LIN {X 0,Y 242.157,Z 688.13,A -85,B 0,C 180,E1 -19275.141,E2 -19275.141} C_VEL
LIN {X 0,Y 242.132,Z 688.251,A -85,B 0,C 180,E1 -19277.962,E2 -19277.962} C_VEL
LIN {X 0,Y 242.388,Z 689.495,A -85,B 0,C 180,E1 -19278.927,E2 -19278.927} C_VEL
LIN {X 0,Y 243.937,Z 692.096,A -85,B 0,C 180,E1 -19280.226,E2 -19280.226} C_VEL
LIN {X 0,Y 247.144,Z 694.46,A -85,B 0,C 180,E1 -19282.354,E2 -19282.354} C_VEL
LIN {X 0,Y 248.695,Z 697.223,A -85,B 0,C 180,E1 -19283.415,E2 -19283.415} C_VEL
LIN {X 0,Y 251.344,Z 699.467,A -85,B 0,C 180,E1 -19284.936,E2 -19284.936} C_VEL
LIN {X 0,Y 251.99,Z 700.132,A -85,B 0,C 180,E1 -19285.297,E2 -19285.297} C_VEL
LIN {X 0,Y 254.265,Z 703.466,A -85,B 0,C 180,E1 -19286.578,E2 -19286.578} C_VEL
LIN {X 0,Y 256.336,Z 705.417,A -85,B 0,C 180,E1 -19287.614,E2 -19287.614} C_VEL
LIN {X 0,Y 258.924,Z 709,A -85,B 0,C 180,E1 -19288.902,E2 -19288.902} C_VEL
LIN {X 0,Y 260.57,Z 710.773,A -85,B 0,C 180,E1 -19289.653,E2 -19289.653} C_VEL
LIN {X 0,Y 263.605,Z 714.655,A -85,B 0,C 180,E1 -19291.005,E2 -19291.005} C_VEL
LIN {X 0,Y 268.675,Z 721.325,A -85,B 0,C 180,E1 -19293.096,E2 -19293.096} C_VEL
LIN {X 0,Y 274.488,Z 729.289,A -85,B 0,C 180,E1 -19295.284,E2 -19295.284} C_VEL
LIN {X 0,Y 282.608,Z 739.443,A -85,B 0,C 180,E1 -19297.978,E2 -19297.978} C_VEL
LIN {X 0,Y 289.117,Z 746.316,A -85,B 0,C 180,E1 -19299.876,E2 -19299.876} C_VEL
LIN {X 0,Y 295.999,Z 752.863,A -85,B 0,C 180,E1 -19301.77,E2 -19301.77} C_VEL
LIN {X 0,Y 303.891,Z 760.01,A -85,B 0,C 180,E1 -19304.075,E2 -19304.075} C_VEL
LIN {X 0,Y 310.616,Z 766.219,A -85,B 0,C 180,E1 -19306.257,E2 -19306.257} C_VEL
LIN {X 0,Y 315.212,Z 770.613,A -85,B 0,C 180,E1 -19307.861,E2 -19307.861} C_VEL
LIN {X 0,Y 320.254,Z 775.282,A -85,B 0,C 180,E1 -19309.758,E2 -19309.758} C_VEL
LIN {X 0,Y 324.928,Z 779.703,A -85,B 0,C 180,E1 -19311.577,E2 -19311.577} C_VEL
LIN {X 0,Y 331.646,Z 785.986,A -85,B 0,C 180,E1 -19314.299,E2 -19314.299} C_VEL
LIN {X 0,Y 335.101,Z 788.959,A -85,B 0,C 180,E1 -19315.743,E2 -19315.743} C_VEL
LIN {X 0,Y 339.882,Z 793.294,A -85,B 0,C 180,E1 -19317.84,E2 -19317.84} C_VEL
LIN {X 0,Y 342.588,Z 795.61,A -85,B 0,C 180,E1 -19319.063,E2 -19319.063} C_VEL
LIN {X 0,Y 346.939,Z 799.679,A -85,B 0,C 180,E1 -19321.138,E2 -19321.138} C_VEL
LIN {X 0,Y 350.25,Z 802.241,A -85,B 0,C 180,E1 -19322.766,E2 -19322.766} C_VEL
LIN {X 0,Y 354.173,Z 806.047,A -85,B 0,C 180,E1 -19324.874,E2 -19324.874} C_VEL
LIN {X 0,Y 358.316,Z 808.916,A -85,B 0,C 180,E1 -19327.197,E2 -19327.197} C_VEL
LIN {X 0,Y 362.043,Z 812.548,A -85,B 0,C 180,E1 -19329.549,E2 -19329.549} C_VEL
LIN {X 0,Y 365.412,Z 815.149,A -85,B 0,C 180,E1 -19331.879,E2 -19331.879} C_VEL
LIN {X 0,Y 368.034,Z 816.748,A -85,B 0,C 180,E1 -19333.849,E2 -19333.849} C_VEL
LIN {X 0,Y 370.527,Z 819.505,A -85,B 0,C 180,E1 -19336.116,E2 -19336.116} C_VEL
LIN {X 0,Y 372.638,Z 821.265,A -85,B 0,C 180,E1 -19338.265,E2 -19338.265} C_VEL
LIN {X 0,Y 374.725,Z 822.511,A -85,B 0,C 180,E1 -19340.809,E2 -19340.809} C_VEL
LIN {X 0,Y 376.488,Z 823.27,A -85,B 0,C 180,E1 -19343.569,E2 -19343.569} C_VEL
LIN {X 0,Y 377.368,Z 823.891,A -85,B 0,C 180,E1 -19345.728,E2 -19345.728} C_VEL
LIN {X 0,Y 377.945,Z 824.103,A -85,B 0,C 180,E1 -19347.869,E2 -19347.869} C_VEL
LIN {X 0,Y 378.148,Z 824.189,A -85,B 0,C 180,E1 -19350,E2 -19350} C_VEL
LIN {X 0,Y 377.944,Z 824.103,A -85,B 0,C 180,E1 -19352.131,E2 -19352.131} C_VEL
LIN {X 0,Y 377.224,Z 823.763,A -85,B 0,C 180,E1 -19354.726,E2 -19354.726} C_VEL
LIN {X 0,Y 376.149,Z 823.23,A -85,B 0,C 180,E1 -19357.007,E2 -19357.007} C_VEL
LIN {X 0,Y 374.33,Z 822.343,A -85,B 0,C 180,E1 -19359.728,E2 -19359.728} C_VEL
LIN {X 0,Y 372.272,Z 820.983,A -85,B 0,C 180,E1 -19362.116,E2 -19362.116} C_VEL
LIN {X 0,Y 369.742,Z 818.743,A -85,B 0,C 180,E1 -19364.631,E2 -19364.631} C_VEL
LIN {X 0,Y 367.379,Z 816.172,A -85,B 0,C 180,E1 -19366.675,E2 -19366.675} C_VEL
LIN {X 0,Y 364.338,Z 814.395,A -85,B 0,C 180,E1 -19368.887,E2 -19368.887} C_VEL
LIN {X 0,Y 360.667,Z 811.337,A -85,B 0,C 180,E1 -19371.326,E2 -19371.326} C_VEL
LIN {X 0,Y 358.319,Z 808.877,A -85,B 0,C 180,E1 -19372.804,E2 -19372.804} C_VEL
LIN {X 0,Y 354.175,Z 806.027,A -85,B 0,C 180,E1 -19375.126,E2 -19375.126} C_VEL
LIN {X 0,Y 350.048,Z 802.014,A -85,B 0,C 180,E1 -19377.342,E2 -19377.342} C_VEL
LIN {X 0,Y 344.973,Z 797.984,A -85,B 0,C 180,E1 -19379.811,E2 -19379.811} C_VEL
LIN {X 0,Y 340.836,Z 794.05,A -85,B 0,C 180,E1 -19381.732,E2 -19381.732} C_VEL
LIN {X 0,Y 335.827,Z 789.683,A -85,B 0,C 180,E1 -19383.943,E2 -19383.943} C_VEL
LIN {X 0,Y 332.449,Z 786.584,A -85,B 0,C 180,E1 -19385.377,E2 -19385.377} C_VEL
LIN {X 0,Y 327.426,Z 782.051,A -85,B 0,C 180,E1 -19387.423,E2 -19387.423} C_VEL
LIN {X 0,Y 324.201,Z 779.091,A -85,B 0,C 180,E1 -19388.703,E2 -19388.703} C_VEL
LIN {X 0,Y 319.113,Z 774.042,A -85,B 0,C 180,E1 -19390.689,E2 -19390.689} C_VEL
LIN {X 0,Y 314.019,Z 769.41,A -85,B 0,C 180,E1 -19392.567,E2 -19392.567} C_VEL
LIN {X 0,Y 309.624,Z 765.385,A -85,B 0,C 180,E1 -19394.072,E2 -19394.072} C_VEL
LIN {X 0,Y 303.772,Z 759.909,A -85,B 0,C 180,E1 -19395.962,E2 -19395.962} C_VEL
LIN {X 0,Y 298.163,Z 754.652,A -85,B 0,C 180,E1 -19397.626,E2 -19397.626} C_VEL
LIN {X 0,Y 291.81,Z 748.998,A -85,B 0,C 180,E1 -19399.386,E2 -19399.386} C_VEL
LIN {X 0,Y 283.81,Z 740.718,A -85,B 0,C 180,E1 -19401.658,E2 -19401.658} C_VEL
LIN {X 0,Y 278.243,Z 734.184,A -85,B 0,C 180,E1 -19403.421,E2 -19403.421} C_VEL
LIN {X 0,Y 269.096,Z 721.878,A -85,B 0,C 180,E1 -19406.739,E2 -19406.739} C_VEL
LIN {X 0,Y 266.598,Z 718.603,A -85,B 0,C 180,E1 -19407.736,E2 -19407.736} C_VEL
LIN {X 0,Y 263.457,Z 714.51,A -85,B 0,C 180,E1 -19409.057,E2 -19409.057} C_VEL
LIN {X 0,Y 260.385,Z 710.48,A -85,B 0,C 180,E1 -19410.435,E2 -19410.435} C_VEL
LIN {X 0,Y 256.965,Z 706.492,A -85,B 0,C 180,E1 -19412.054,E2 -19412.054} C_VEL
LIN {X 0,Y 255.896,Z 704.836,A -85,B 0,C 180,E1 -19412.612,E2 -19412.612} C_VEL
LIN {X 0,Y 253.226,Z 702.224,A -85,B 0,C 180,E1 -19413.979,E2 -19413.979} C_VEL
LIN {X 0,Y 251.561,Z 699.597,A -85,B 0,C 180,E1 -19414.948,E2 -19414.948} C_VEL
LIN {X 0,Y 248.847,Z 697.414,A -85,B 0,C 180,E1 -19416.49,E2 -19416.49} C_VEL
LIN {X 0,Y 246.704,Z 693.991,A -85,B 0,C 180,E1 -19417.934,E2 -19417.934} C_VEL
LIN {X 0,Y 243.937,Z 692.096,A -85,B 0,C 180,E1 -19419.774,E2 -19419.774} C_VEL
LIN {X 0,Y 242.353,Z 689.417,A -85,B 0,C 180,E1 -19421.125,E2 -19421.125} C_VEL
LIN {X 0,Y 242.133,Z 688.246,A -85,B 0,C 180,E1 -19422.093,E2 -19422.093} C_VEL
LIN {X 0,Y 242.156,Z 688.106,A -85,B 0,C 180,E1 -19426.575,E2 -19426.575} C_VEL
LIN {X 0,Y 242.419,Z 688.073,A -85,B 0,C 180,E1 -19431.666,E2 -19431.666} C_VEL
LIN {X 0,Y 242.256,Z 688.12,A -85,B 0,C 180,E1 -19435.008,E2 -19435.008} C_VEL
LIN {X 0,Y 242.631,Z 688.05,A -85,B 0,C 180,E1 -19438.341,E2 -19438.341} C_VEL
LIN {X 0,Y 242.631,Z 688.052,A -85,B 0,C 180,E1 -19441.66,E2 -19441.66} C_VEL
LIN {X 0,Y 242.427,Z 688.078,A -85,B 0,C 180,E1 -19446.659,E2 -19446.659} C_VEL
LIN {X 0,Y 242.309,Z 688.104,A -85,B 0,C 180,E1 -19450.022,E2 -19450.022} C_VEL
LIN {X 0,Y 242.151,Z 688.127,A -85,B 0,C 180,E1 -19455.142,E2 -19455.142} C_VEL
LIN {X 0,Y 242.154,Z 688.429,A -85,B 0,C 180,E1 -19457.743,E2 -19457.743} C_VEL
LIN {X 0,Y 242.453,Z 689.706,A -85,B 0,C 180,E1 -19458.594,E2 -19458.594} C_VEL
LIN {X 0,Y 243.896,Z 692.084,A -85,B 0,C 180,E1 -19459.791,E2 -19459.791} C_VEL
LIN {X 0,Y 246.644,Z 693.971,A -85,B 0,C 180,E1 -19461.623,E2 -19461.623} C_VEL
LIN {X 0,Y 247.502,Z 695.283,A -85,B 0,C 180,E1 -19462.211,E2 -19462.211} C_VEL
LIN {X 0,Y 249.266,Z 697.887,A -85,B 0,C 180,E1 -19463.359,E2 -19463.359} C_VEL
LIN {X 0,Y 251.914,Z 700.026,A -85,B 0,C 180,E1 -19464.846,E2 -19464.846} C_VEL
LIN {X 0,Y 254.117,Z 703.305,A -85,B 0,C 180,E1 -19466.094,E2 -19466.094} C_VEL
LIN {X 0,Y 256.371,Z 705.449,A -85,B 0,C 180,E1 -19467.224,E2 -19467.224} C_VEL
LIN {X 0,Y 259.014,Z 709.076,A -85,B 0,C 180,E1 -19468.535,E2 -19468.535} C_VEL
LIN {X 0,Y 260.601,Z 710.841,A -85,B 0,C 180,E1 -19469.262,E2 -19469.262} C_VEL
LIN {X 0,Y 263.715,Z 714.755,A -85,B 0,C 180,E1 -19470.643,E2 -19470.643} C_VEL
LIN {X 0,Y 268.241,Z 721.279,A -85,B 0,C 180,E1 -19472.543,E2 -19472.543} C_VEL
LIN {X 0,Y 272.38,Z 727.881,A -85,B 0,C 180,E1 -19474.176,E2 -19474.176} C_VEL
LIN {X 0,Y 279.24,Z 739.541,A -85,B 0,C 180,E1 -19476.675,E2 -19476.675} C_VEL
LIN {X 0,Y 286.08,Z 752.594,A -85,B 0,C 180,E1 -19478.974,E2 -19478.974} C_VEL
LIN {X 0,Y 292.085,Z 765.049,A -85,B 0,C 180,E1 -19480.857,E2 -19480.857} C_VEL
LIN {X 0,Y 296.083,Z 774.289,A -85,B 0,C 180,E1 -19482.065,E2 -19482.065} C_VEL
LIN {X 0,Y 295.264,Z 789.935,A -85,B 0,C 180,E1 -19482.443,E2 -19482.443} C_VEL
LIN {X 0,Y 294.474,Z 795.788,A -85,B 0,C 180,E1 -19482.482,E2 -19482.482} C_VEL
LIN {X 0,Y 289.416,Z 814.875,A -85,B 0,C 180,E1 -19482.08,E2 -19482.08} C_VEL
LIN {X 0,Y 288.604,Z 820.73,A -85,B 0,C 180,E1 -19482.114,E2 -19482.114} C_VEL
LIN {X 0,Y 284.395,Z 890.144,A -85,B 0,C 180,E1 -19483.772,E2 -19483.772} C_VEL
LIN {X 0,Y 283.091,Z 902.745,A -85,B 0,C 180,E1 -19484.196,E2 -19484.196} C_VEL
LIN {X 0,Y 281.233,Z 915.218,A -85,B 0,C 180,E1 -19484.73,E2 -19484.73} C_VEL
LIN {X 0,Y 278.913,Z 927.393,A -85,B 0,C 180,E1 -19485.382,E2 -19485.382} C_VEL
LIN {X 0,Y 276.549,Z 938.778,A -85,B 0,C 180,E1 -19486.172,E2 -19486.172} C_VEL
LIN {X 0,Y 273.265,Z 952.009,A -85,B 0,C 180,E1 -19487.288,E2 -19487.288} C_VEL
LIN {X 0,Y 270.044,Z 963.302,A -85,B 0,C 180,E1 -19488.423,E2 -19488.423} C_VEL
LIN {X 0,Y 266.166,Z 975.709,A -85,B 0,C 180,E1 -19489.935,E2 -19489.935} C_VEL
LIN {X 0,Y 262.462,Z 986.529,A -85,B 0,C 180,E1 -19491.497,E2 -19491.497} C_VEL
LIN {X 0,Y 258.484,Z 997.021,A -85,B 0,C 180,E1 -19493.263,E2 -19493.263} C_VEL
LIN {X 0,Y 254.908,Z 1006.289,A -85,B 0,C 180,E1 -19495.105,E2 -19495.105} C_VEL
LIN {X 0,Y 250.75,Z 1016.429,A -85,B 0,C 180,E1 -19497.482,E2 -19497.482} C_VEL
LIN {X 0,Y 247.32,Z 1024.542,A -85,B 0,C 180,E1 -19499.71,E2 -19499.71} C_VEL
LIN {X 0,Y 243.66,Z 1033.143,A -85,B 0,C 180,E1 -19502.517,E2 -19502.517} C_VEL
LIN {X 0,Y 240.85,Z 1039.875,A -85,B 0,C 180,E1 -19505.114,E2 -19505.114} C_VEL
LIN {X 0,Y 238.008,Z 1046.841,A -85,B 0,C 180,E1 -19508.34,E2 -19508.34} C_VEL
LIN {X 0,Y 236.243,Z 1051.496,A -85,B 0,C 180,E1 -19510.899,E2 -19510.899} C_VEL
LIN {X 0,Y 234.564,Z 1056.604,A -85,B 0,C 180,E1 -19514.357,E2 -19514.357} C_VEL
LIN {X 0,Y 233.371,Z 1060.609,A -85,B 0,C 180,E1 -19517.831,E2 -19517.831} C_VEL
LIN {X 0,Y 232.842,Z 1063.577,A -85,B 0,C 180,E1 -19521.32,E2 -19521.32} C_VEL
LIN {X 0,Y 232.7,Z 1064.768,A -85,B 0,C 180,E1 -19523.061,E2 -19523.061} C_VEL
LIN {X 0,Y 232.651,Z 1066.246,A -85,B 0,C 180,E1 -19526.536,E2 -19526.536} C_VEL
LIN {X 0,Y 232.801,Z 1066.741,A -85,B 0,C 180,E1 -19530,E2 -19530} C_VEL
LIN {X 0,Y 232.651,Z 1066.246,A -85,B 0,C 180,E1 -19533.464,E2 -19533.464} C_VEL
LIN {X 0,Y 232.7,Z 1064.768,A -85,B 0,C 180,E1 -19536.939,E2 -19536.939} C_VEL
LIN {X 0,Y 233.04,Z 1062.289,A -85,B 0,C 180,E1 -19540.425,E2 -19540.425} C_VEL
LIN {X 0,Y 234.206,Z 1057.693,A -85,B 0,C 180,E1 -19544.777,E2 -19544.777} C_VEL
LIN {X 0,Y 235.787,Z 1052.848,A -85,B 0,C 180,E1 -19548.238,E2 -19548.238} C_VEL
LIN {X 0,Y 237.391,Z 1048.465,A -85,B 0,C 180,E1 -19550.809,E2 -19550.809} C_VEL
LIN {X 0,Y 239.44,Z 1043.402,A -85,B 0,C 180,E1 -19553.343,E2 -19553.343} C_VEL
LIN {X 0,Y 242.248,Z 1036.477,A -85,B 0,C 180,E1 -19556.258,E2 -19556.258} C_VEL
LIN {X 0,Y 245.703,Z 1028.382,A -85,B 0,C 180,E1 -19559.094,E2 -19559.094} C_VEL
LIN {X 0,Y 249.164,Z 1020.417,A -85,B 0,C 180,E1 -19561.453,E2 -19561.453} C_VEL
LIN {X 0,Y 252.896,Z 1011.305,A -85,B 0,C 180,E1 -19563.765,E2 -19563.765} C_VEL
LIN {X 0,Y 256.333,Z 1002.739,A -85,B 0,C 180,E1 -19565.634,E2 -19565.634} C_VEL
LIN {X 0,Y 260.727,Z 990.874,A -85,B 0,C 180,E1 -19567.823,E2 -19567.823} C_VEL
LIN {X 0,Y 264.497,Z 980.719,A -85,B 0,C 180,E1 -19569.373,E2 -19569.373} C_VEL
LIN {X 0,Y 268.315,Z 969.054,A -85,B 0,C 180,E1 -19570.905,E2 -19570.905} C_VEL
LIN {X 0,Y 271.869,Z 957.033,A -85,B 0,C 180,E1 -19572.229,E2 -19572.229} C_VEL
LIN {X 0,Y 275.13,Z 944.719,A -85,B 0,C 180,E1 -19573.352,E2 -19573.352} C_VEL
LIN {X 0,Y 277.951,Z 932.178,A -85,B 0,C 180,E1 -19574.305,E2 -19574.305} C_VEL
LIN {X 0,Y 280.57,Z 918.763,A -85,B 0,C 180,E1 -19575.104,E2 -19575.104} C_VEL
LIN {X 0,Y 282.658,Z 905.869,A -85,B 0,C 180,E1 -19575.691,E2 -19575.691} C_VEL
LIN {X 0,Y 284.256,Z 892.458,A -85,B 0,C 180,E1 -19576.149,E2 -19576.149} C_VEL
LIN {X 0,Y 285.97,Z 865.198,A -85,B 0,C 180,E1 -19576.851,E2 -19576.851} C_VEL
LIN {X 0,Y 291.182,Z 777.985,A -85,B 0,C 180,E1 -19578.872,E2 -19578.872} C_VEL
LIN {X 0,Y 291.068,Z 776.493,A -85,B 0,C 180,E1 -19578.952,E2 -19578.952} C_VEL
LIN {X 0,Y 285.259,Z 763.336,A -85,B 0,C 180,E1 -19580.809,E2 -19580.809} C_VEL
LIN {X 0,Y 278.575,Z 749.866,A -85,B 0,C 180,E1 -19583.074,E2 -19583.074} C_VEL
LIN {X 0,Y 273.098,Z 739.77,A -85,B 0,C 180,E1 -19585.069,E2 -19585.069} C_VEL
LIN {X 0,Y 266.936,Z 729.437,A -85,B 0,C 180,E1 -19587.495,E2 -19587.495} C_VEL
LIN {X 0,Y 263.033,Z 723.353,A -85,B 0,C 180,E1 -19589.158,E2 -19589.158} C_VEL
LIN {X 0,Y 260.683,Z 720.268,A -85,B 0,C 180,E1 -19590.193,E2 -19590.193} C_VEL
LIN {X 0,Y 257.341,Z 715.903,A -85,B 0,C 180,E1 -19591.757,E2 -19591.757} C_VEL
LIN {X 0,Y 254.259,Z 711.919,A -85,B 0,C 180,E1 -19593.309,E2 -19593.309} C_VEL
LIN {X 0,Y 250.599,Z 707.706,A -85,B 0,C 180,E1 -19595.289,E2 -19595.289} C_VEL
LIN {X 0,Y 249.582,Z 706.174,A -85,B 0,C 180,E1 -19595.901,E2 -19595.901} C_VEL
LIN {X 0,Y 246.769,Z 703.584,A -85,B 0,C 180,E1 -19597.581,E2 -19597.581} C_VEL
LIN {X 0,Y 245.071,Z 700.739,A -85,B 0,C 180,E1 -19598.777,E2 -19598.777} C_VEL
LIN {X 0,Y 242.377,Z 698.784,A -85,B 0,C 180,E1 -19600.631,E2 -19600.631} C_VEL
LIN {X 0,Y 240.648,Z 695.967,A -85,B 0,C 180,E1 -19602.087,E2 -19602.087} C_VEL
LIN {X 0,Y 239.897,Z 694.934,A -85,B 0,C 180,E1 -19602.745,E2 -19602.745} C_VEL
LIN {X 0,Y 236.953,Z 692.981,A -85,B 0,C 180,E1 -19605.397,E2 -19605.397} C_VEL
LIN {X 0,Y 235.329,Z 690.078,A -85,B 0,C 180,E1 -19607.495,E2 -19607.495} C_VEL
LIN {X 0,Y 235.168,Z 689.024,A -85,B 0,C 180,E1 -19608.962,E2 -19608.962} C_VEL
LIN {X 0,Y 235.371,Z 688.951,A -85,B 0,C 180,E1 -19611.413,E2 -19611.413} C_VEL
LIN {X 0,Y 235.398,Z 688.95,A -85,B 0,C 180,E1 -19613.141,E2 -19613.141} C_VEL
LIN {X 0,Y 235.59,Z 688.926,A -85,B 0,C 180,E1 -19618.29,E2 -19618.29} C_VEL
LIN {X 0,Y 235.59,Z 688.925,A -85,B 0,C 180,E1 -19621.709,E2 -19621.709} C_VEL
LIN {X 0,Y 235.397,Z 688.951,A -85,B 0,C 180,E1 -19626.858,E2 -19626.858} C_VEL
LIN {X 0,Y 235.232,Z 689.005,A -85,B 0,C 180,E1 -19630.326,E2 -19630.326} C_VEL
LIN {X 0,Y 235.194,Z 689.499,A -85,B 0,C 180,E1 -19632.292,E2 -19632.292} C_VEL
LIN {X 0,Y 235.642,Z 690.924,A -85,B 0,C 180,E1 -19633.474,E2 -19633.474} C_VEL
LIN {X 0,Y 237.185,Z 693.203,A -85,B 0,C 180,E1 -19635.246,E2 -19635.246} C_VEL
LIN {X 0,Y 240.413,Z 695.413,A -85,B 0,C 180,E1 -19638.095,E2 -19638.095} C_VEL
LIN {X 0,Y 242.289,Z 698.654,A -85,B 0,C 180,E1 -19639.706,E2 -19639.706} C_VEL
LIN {X 0,Y 244.989,Z 700.698,A -85,B 0,C 180,E1 -19641.578,E2 -19641.578} C_VEL
LIN {X 0,Y 247.688,Z 704.621,A -85,B 0,C 180,E1 -19643.405,E2 -19643.405} C_VEL
LIN {X 0,Y 250.035,Z 706.686,A -85,B 0,C 180,E1 -19644.77,E2 -19644.77} C_VEL
LIN {X 0,Y 252.548,Z 710.161,A -85,B 0,C 180,E1 -19646.21,E2 -19646.21} C_VEL
LIN {X 0,Y 254.313,Z 712.015,A -85,B 0,C 180,E1 -19647.127,E2 -19647.127} C_VEL
LIN {X 0,Y 257.121,Z 715.679,A -85,B 0,C 180,E1 -19648.546,E2 -19648.546} C_VEL
LIN {X 0,Y 258.462,Z 717.383,A -85,B 0,C 180,E1 -19649.188,E2 -19649.188} C_VEL
LIN {X 0,Y 262.751,Z 722.957,A -85,B 0,C 180,E1 -19651.126,E2 -19651.126} C_VEL
LIN {X 0,Y 266.457,Z 727.884,A -85,B 0,C 180,E1 -19652.675,E2 -19652.675} C_VEL
LIN {X 0,Y 279.488,Z 745.151,A -85,B 0,C 180,E1 -19657.384,E2 -19657.384} C_VEL
LIN {X 0,Y 286.696,Z 752.785,A -85,B 0,C 180,E1 -19659.54,E2 -19659.54} C_VEL
LIN {X 0,Y 293.599,Z 759.313,A -85,B 0,C 180,E1 -19661.43,E2 -19661.43} C_VEL
LIN {X 0,Y 300.628,Z 765.685,A -85,B 0,C 180,E1 -19663.455,E2 -19663.455} C_VEL
LIN {X 0,Y 304.805,Z 769.406,A -85,B 0,C 180,E1 -19664.728,E2 -19664.728} C_VEL
LIN {X 0,Y 309.685,Z 773.681,A -85,B 0,C 180,E1 -19666.306,E2 -19666.306} C_VEL
LIN {X 0,Y 315.306,Z 779.062,A -85,B 0,C 180,E1 -19668.282,E2 -19668.282} C_VEL
LIN {X 0,Y 319.999,Z 783.569,A -85,B 0,C 180,E1 -19670.062,E2 -19670.062} C_VEL
LIN {X 0,Y 325.699,Z 788.7,A -85,B 0,C 180,E1 -19672.28,E2 -19672.28} C_VEL
LIN {X 0,Y 330.659,Z 793.216,A -85,B 0,C 180,E1 -19674.297,E2 -19674.297} C_VEL
LIN {X 0,Y 333.474,Z 795.703,A -85,B 0,C 180,E1 -19675.473,E2 -19675.473} C_VEL
LIN {X 0,Y 338.278,Z 800.003,A -85,B 0,C 180,E1 -19677.547,E2 -19677.547} C_VEL
LIN {X 0,Y 340.875,Z 802.2,A -85,B 0,C 180,E1 -19678.714,E2 -19678.714} C_VEL
LIN {X 0,Y 345.38,Z 806.398,A -85,B 0,C 180,E1 -19680.847,E2 -19680.847} C_VEL
LIN {X 0,Y 348.716,Z 808.932,A -85,B 0,C 180,E1 -19682.469,E2 -19682.469} C_VEL
LIN {X 0,Y 352.697,Z 812.745,A -85,B 0,C 180,E1 -19684.577,E2 -19684.577} C_VEL
LIN {X 0,Y 356.872,Z 815.691,A -85,B 0,C 180,E1 -19686.88,E2 -19686.88} C_VEL
LIN {X 0,Y 360.806,Z 819.411,A -85,B 0,C 180,E1 -19689.334,E2 -19689.334} C_VEL
LIN {X 0,Y 364.226,Z 822.049,A -85,B 0,C 180,E1 -19691.676,E2 -19691.676} C_VEL
LIN {X 0,Y 366.994,Z 823.751,A -85,B 0,C 180,E1 -19693.725,E2 -19693.725} C_VEL
LIN {X 0,Y 369.473,Z 826.446,A -85,B 0,C 180,E1 -19695.952,E2 -19695.952} C_VEL
LIN {X 0,Y 371.492,Z 828.14,A -85,B 0,C 180,E1 -19697.989,E2 -19697.989} C_VEL
LIN {X 0,Y 373.441,Z 829.38,A -85,B 0,C 180,E1 -19700.249,E2 -19700.249} C_VEL
LIN {X 0,Y 375.282,Z 830.27,A -85,B 0,C 180,E1 -19702.993,E2 -19702.993} C_VEL
LIN {X 0,Y 376.498,Z 830.932,A -85,B 0,C 180,E1 -19705.718,E2 -19705.718} C_VEL
LIN {X 0,Y 377.076,Z 831.149,A -85,B 0,C 180,E1 -19707.864,E2 -19707.864} C_VEL
LIN {X 0,Y 377.283,Z 831.235,A -85,B 0,C 180,E1 -19710,E2 -19710} C_VEL
LIN {X 0,Y 377.076,Z 831.148,A -85,B 0,C 180,E1 -19712.136,E2 -19712.136} C_VEL
LIN {X 0,Y 376.354,Z 830.811,A -85,B 0,C 180,E1 -19714.737,E2 -19714.737} C_VEL
LIN {X 0,Y 375.104,Z 830.173,A -85,B 0,C 180,E1 -19717.299,E2 -19717.299} C_VEL
LIN {X 0,Y 373.441,Z 829.385,A -85,B 0,C 180,E1 -19719.751,E2 -19719.751} C_VEL
LIN {X 0,Y 371.365,Z 828.015,A -85,B 0,C 180,E1 -19722.146,E2 -19722.146} C_VEL
LIN {X 0,Y 368.91,Z 825.922,A -85,B 0,C 180,E1 -19724.58,E2 -19724.58} C_VEL
LIN {X 0,Y 366.201,Z 823.109,A -85,B 0,C 180,E1 -19726.89,E2 -19726.89} C_VEL
LIN {X 0,Y 362.98,Z 821.155,A -85,B 0,C 180,E1 -19729.217,E2 -19729.217} C_VEL
LIN {X 0,Y 359.096,Z 817.848,A -85,B 0,C 180,E1 -19731.759,E2 -19731.759} C_VEL
LIN {X 0,Y 356.973,Z 815.726,A -85,B 0,C 180,E1 -19733.061,E2 -19733.061} C_VEL
LIN {X 0,Y 352.563,Z 812.65,A -85,B 0,C 180,E1 -19735.495,E2 -19735.495} C_VEL
LIN {X 0,Y 347.543,Z 807.97,A -85,B 0,C 180,E1 -19738.112,E2 -19738.112} C_VEL
LIN {X 0,Y 343.037,Z 804.349,A -85,B 0,C 180,E1 -19740.266,E2 -19740.266} C_VEL
LIN {X 0,Y 339.196,Z 800.725,A -85,B 0,C 180,E1 -19742.037,E2 -19742.037} C_VEL
LIN {X 0,Y 334.098,Z 796.312,A -85,B 0,C 180,E1 -19744.261,E2 -19744.261} C_VEL
LIN {X 0,Y 330.812,Z 793.323,A -85,B 0,C 180,E1 -19745.642,E2 -19745.642} C_VEL
LIN {X 0,Y 325.496,Z 788.535,A -85,B 0,C 180,E1 -19747.801,E2 -19747.801} C_VEL
LIN {X 0,Y 318.755,Z 782.313,A -85,B 0,C 180,E1 -19750.423,E2 -19750.423} C_VEL
LIN {X 0,Y 315.079,Z 778.87,A -85,B 0,C 180,E1 -19751.799,E2 -19751.799} C_VEL
LIN {X 0,Y 308.446,Z 772.688,A -85,B 0,C 180,E1 -19754.104,E2 -19754.104} C_VEL
LIN {X 0,Y 301.432,Z 766.329,A -85,B 0,C 180,E1 -19756.309,E2 -19756.309} C_VEL
LIN {X 0,Y 296.413,Z 761.822,A -85,B 0,C 180,E1 -19757.777,E2 -19757.777} C_VEL
LIN {X 0,Y 288.735,Z 754.866,A -85,B 0,C 180,E1 -19759.89,E2 -19759.89} C_VEL
LIN {X 0,Y 281.034,Z 746.827,A -85,B 0,C 180,E1 -19762.134,E2 -19762.134} C_VEL
LIN {X 0,Y 275.221,Z 739.886,A -85,B 0,C 180,E1 -19764.033,E2 -19764.033} C_VEL
LIN {X 0,Y 264.577,Z 725.223,A -85,B 0,C 180,E1 -19768.105,E2 -19768.105} C_VEL
LIN {X 0,Y 260.8,Z 720.394,A -85,B 0,C 180,E1 -19769.735,E2 -19769.735} C_VEL
LIN {X 0,Y 257.235,Z 715.776,A -85,B 0,C 180,E1 -19771.401,E2 -19771.401} C_VEL
LIN {X 0,Y 254.398,Z 712.153,A -85,B 0,C 180,E1 -19772.827,E2 -19772.827} C_VEL
LIN {X 0,Y 253.263,Z 710.813,A -85,B 0,C 180,E1 -19773.419,E2 -19773.419} C_VEL
LIN {X 0,Y 250.554,Z 707.612,A -85,B 0,C 180,E1 -19774.91,E2 -19774.91} C_VEL
LIN {X 0,Y 249.639,Z 706.166,A -85,B 0,C 180,E1 -19775.465,E2 -19775.465} C_VEL
LIN {X 0,Y 246.853,Z 703.681,A -85,B 0,C 180,E1 -19777.121,E2 -19777.121} C_VEL
LIN {X 0,Y 244.989,Z 700.698,A -85,B 0,C 180,E1 -19778.422,E2 -19778.422} C_VEL
LIN {X 0,Y 242.291,Z 698.641,A -85,B 0,C 180,E1 -19780.294,E2 -19780.294} C_VEL
LIN {X 0,Y 240.575,Z 695.76,A -85,B 0,C 180,E1 -19781.753,E2 -19781.753} C_VEL
LIN {X 0,Y 239.683,Z 694.844,A -85,B 0,C 180,E1 -19782.51,E2 -19782.51} C_VEL
LIN {X 0,Y 236.785,Z 692.785,A -85,B 0,C 180,E1 -19785.168,E2 -19785.168} C_VEL
LIN {X 0,Y 235.347,Z 690.143,A -85,B 0,C 180,E1 -19787.058,E2 -19787.058} C_VEL
LIN {X 0,Y 235.176,Z 689.072,A -85,B 0,C 180,E1 -19788.582,E2 -19788.582} C_VEL
LIN {X 0,Y 235.369,Z 688.952,A -85,B 0,C 180,E1 -19791.414,E2 -19791.414} C_VEL
LIN {X 0,Y 235.396,Z 688.949,A -85,B 0,C 180,E1 -19793.142,E2 -19793.142} C_VEL
LIN {X 0,Y 235.59,Z 688.926,A -85,B 0,C 180,E1 -19798.291,E2 -19798.291} C_VEL
LIN {X 0,Y 235.59,Z 688.928,A -85,B 0,C 180,E1 -19801.71,E2 -19801.71} C_VEL
LIN {X 0,Y 235.398,Z 688.951,A -85,B 0,C 180,E1 -19806.859,E2 -19806.859} C_VEL
LIN {X 0,Y 235.2,Z 689.043,A -85,B 0,C 180,E1 -19810.764,E2 -19810.764} C_VEL
LIN {X 0,Y 235.238,Z 689.626,A -85,B 0,C 180,E1 -19812.072,E2 -19812.072} C_VEL
LIN {X 0,Y 235.938,Z 691.525,A -85,B 0,C 180,E1 -19813.457,E2 -19813.457} C_VEL
LIN {X 0,Y 237.788,Z 693.718,A -85,B 0,C 180,E1 -19815.427,E2 -19815.427} C_VEL
LIN {X 0,Y 240.378,Z 695.377,A -85,B 0,C 180,E1 -19817.658,E2 -19817.658} C_VEL
LIN {X 0,Y 242.119,Z 698.486,A -85,B 0,C 180,E1 -19819.17,E2 -19819.17} C_VEL
LIN {X 0,Y 244.692,Z 700.576,A -85,B 0,C 180,E1 -19820.983,E2 -19820.983} C_VEL
LIN {X 0,Y 245.385,Z 701.183,A -85,B 0,C 180,E1 -19821.444,E2 -19821.444} C_VEL
LIN {X 0,Y 247.178,Z 704.096,A -85,B 0,C 180,E1 -19822.683,E2 -19822.683} C_VEL
LIN {X 0,Y 250.063,Z 706.745,A -85,B 0,C 180,E1 -19824.381,E2 -19824.381} C_VEL
LIN {X 0,Y 252.489,Z 710.106,A -85,B 0,C 180,E1 -19825.772,E2 -19825.772} C_VEL
LIN {X 0,Y 254.343,Z 712.062,A -85,B 0,C 180,E1 -19826.736,E2 -19826.736} C_VEL
LIN {X 0,Y 257.459,Z 716.038,A -85,B 0,C 180,E1 -19828.299,E2 -19828.299} C_VEL
LIN {X 0,Y 262.541,Z 722.671,A -85,B 0,C 180,E1 -19830.627,E2 -19830.627} C_VEL
LIN {X 0,Y 265.549,Z 727.214,A -85,B 0,C 180,E1 -19831.925,E2 -19831.925} C_VEL
LIN {X 0,Y 270.85,Z 735.879,A -85,B 0,C 180,E1 -19834.071,E2 -19834.071} C_VEL
LIN {X 0,Y 277.073,Z 747.03,A -85,B 0,C 180,E1 -19836.393,E2 -19836.393} C_VEL
LIN {X 0,Y 283.438,Z 759.57,A -85,B 0,C 180,E1 -19838.592,E2 -19838.592} C_VEL
LIN {X 0,Y 289.231,Z 772.137,A -85,B 0,C 180,E1 -19840.469,E2 -19840.469} C_VEL
LIN {X 0,Y 291.187,Z 776.785,A -85,B 0,C 180,E1 -19841.085,E2 -19841.085} C_VEL
LIN {X 0,Y 288.604,Z 820.73,A -85,B 0,C 180,E1 -19842.114,E2 -19842.114} C_VEL
LIN {X 0,Y 287.794,Z 826.586,A -85,B 0,C 180,E1 -19842.15,E2 -19842.15} C_VEL
LIN {X 0,Y 282.774,Z 845.685,A -85,B 0,C 180,E1 -19841.738,E2 -19841.738} C_VEL
LIN {X 0,Y 281.985,Z 851.539,A -85,B 0,C 180,E1 -19841.778,E2 -19841.778} C_VEL
LIN {X 0,Y 279.451,Z 890.753,A -85,B 0,C 180,E1 -19842.743,E2 -19842.743} C_VEL
LIN {X 0,Y 278.04,Z 903.623,A -85,B 0,C 180,E1 -19843.188,E2 -19843.188} C_VEL
LIN {X 0,Y 276.08,Z 916.12,A -85,B 0,C 180,E1 -19843.738,E2 -19843.738} C_VEL
LIN {X 0,Y 273.637,Z 928.383,A -85,B 0,C 180,E1 -19844.414,E2 -19844.414} C_VEL
LIN {X 0,Y 270.963,Z 940.552,A -85,B 0,C 180,E1 -19845.29,E2 -19845.29} C_VEL
LIN {X 0,Y 268.073,Z 951.803,A -85,B 0,C 180,E1 -19846.255,E2 -19846.255} C_VEL
LIN {X 0,Y 264.273,Z 964.533,A -85,B 0,C 180,E1 -19847.562,E2 -19847.562} C_VEL
LIN {X 0,Y 260.621,Z 975.811,A -85,B 0,C 180,E1 -19848.965,E2 -19848.965} C_VEL
LIN {X 0,Y 256.922,Z 986.323,A -85,B 0,C 180,E1 -19850.507,E2 -19850.507} C_VEL
LIN {X 0,Y 252.775,Z 996.813,A -85,B 0,C 180,E1 -19852.291,E2 -19852.291} C_VEL
LIN {X 0,Y 249.057,Z 1006.082,A -85,B 0,C 180,E1 -19854.16,E2 -19854.16} C_VEL
LIN {X 0,Y 244.839,Z 1015.845,A -85,B 0,C 180,E1 -19856.47,E2 -19856.47} C_VEL
LIN {X 0,Y 241.125,Z 1024.333,A -85,B 0,C 180,E1 -19858.846,E2 -19858.846} C_VEL
LIN {X 0,Y 237.284,Z 1032.934,A -85,B 0,C 180,E1 -19861.713,E2 -19861.713} C_VEL
LIN {X 0,Y 234.061,Z 1040.26,A -85,B 0,C 180,E1 -19864.636,E2 -19864.636} C_VEL
LIN {X 0,Y 231.333,Z 1046.633,A -85,B 0,C 180,E1 -19867.682,E2 -19867.682} C_VEL
LIN {X 0,Y 229.454,Z 1051.288,A -85,B 0,C 180,E1 -19870.311,E2 -19870.311} C_VEL
LIN {X 0,Y 227.632,Z 1056.395,A -85,B 0,C 180,E1 -19873.867,E2 -19873.867} C_VEL
LIN {X 0,Y 226.366,Z 1060.402,A -85,B 0,C 180,E1 -19877.448,E2 -19877.448} C_VEL
LIN {X 0,Y 225.761,Z 1063.37,A -85,B 0,C 180,E1 -19881.046,E2 -19881.046} C_VEL
LIN {X 0,Y 225.61,Z 1064.562,A -85,B 0,C 180,E1 -19882.842,E2 -19882.842} C_VEL
LIN {X 0,Y 225.549,Z 1066.04,A -85,B 0,C 180,E1 -19886.427,E2 -19886.427} C_VEL
LIN {X 0,Y 225.714,Z 1066.536,A -85,B 0,C 180,E1 -19890,E2 -19890} C_VEL
LIN {X 0,Y 225.554,Z 1065.725,A -85,B 0,C 180,E1 -19894.378,E2 -19894.378} C_VEL
LIN {X 0,Y 225.61,Z 1064.562,A -85,B 0,C 180,E1 -19897.158,E2 -19897.158} C_VEL
LIN {X 0,Y 226.005,Z 1062.082,A -85,B 0,C 180,E1 -19900.753,E2 -19900.753} C_VEL
LIN {X 0,Y 227.264,Z 1057.485,A -85,B 0,C 180,E1 -19905.239,E2 -19905.239} C_VEL
LIN {X 0,Y 228.444,Z 1053.989,A -85,B 0,C 180,E1 -19907.917,E2 -19907.917} C_VEL
LIN {X 0,Y 230.665,Z 1048.256,A -85,B 0,C 180,E1 -19911.445,E2 -19911.445} C_VEL
LIN {X 0,Y 232.826,Z 1043.193,A -85,B 0,C 180,E1 -19914.048,E2 -19914.048} C_VEL
LIN {X 0,Y 235.796,Z 1036.268,A -85,B 0,C 180,E1 -19917.034,E2 -19917.034} C_VEL
LIN {X 0,Y 239.444,Z 1028.174,A -85,B 0,C 180,E1 -19919.931,E2 -19919.931} C_VEL
LIN {X 0,Y 243.025,Z 1020.208,A -85,B 0,C 180,E1 -19922.343,E2 -19922.343} C_VEL
LIN {X 0,Y 246.926,Z 1011.096,A -85,B 0,C 180,E1 -19924.696,E2 -19924.696} C_VEL
LIN {X 0,Y 250.529,Z 1002.531,A -85,B 0,C 180,E1 -19926.591,E2 -19926.591} C_VEL
LIN {X 0,Y 254.692,Z 991.754,A -85,B 0,C 180,E1 -19928.631,E2 -19928.631} C_VEL
LIN {X 0,Y 258.987,Z 980.511,A -85,B 0,C 180,E1 -19930.381,E2 -19930.381} C_VEL
LIN {X 0,Y 262.941,Z 968.847,A -85,B 0,C 180,E1 -19931.928,E2 -19931.928} C_VEL
LIN {X 0,Y 266.629,Z 956.827,A -85,B 0,C 180,E1 -19933.26,E2 -19933.26} C_VEL
LIN {X 0,Y 270.002,Z 944.513,A -85,B 0,C 180,E1 -19934.389,E2 -19934.389} C_VEL
LIN {X 0,Y 272.913,Z 931.972,A -85,B 0,C 180,E1 -19935.347,E2 -19935.347} C_VEL
LIN {X 0,Y 275.564,Z 918.788,A -85,B 0,C 180,E1 -19936.138,E2 -19936.138} C_VEL
LIN {X 0,Y 277.751,Z 905.559,A -85,B 0,C 180,E1 -19936.744,E2 -19936.744} C_VEL
LIN {X 0,Y 279.398,Z 891.997,A -85,B 0,C 180,E1 -19937.208,E2 -19937.208} C_VEL
LIN {X 0,Y 281.266,Z 863.199,A -85,B 0,C 180,E1 -19937.949,E2 -19937.949} C_VEL
LIN {X 0,Y 286.465,Z 779.471,A -85,B 0,C 180,E1 -19939.9,E2 -19939.9} C_VEL
LIN {X 0,Y 280.611,Z 766.179,A -85,B 0,C 180,E1 -19941.864,E2 -19941.864} C_VEL
LIN {X 0,Y 273.658,Z 751.997,A -85,B 0,C 180,E1 -19944.362,E2 -19944.362} C_VEL
LIN {X 0,Y 267.265,Z 740.413,A -85,B 0,C 180,E1 -19946.856,E2 -19946.856} C_VEL
LIN {X 0,Y 261.559,Z 730.904,A -85,B 0,C 180,E1 -19949.301,E2 -19949.301} C_VEL
LIN {X 0,Y 258.357,Z 726.484,A -85,B 0,C 180,E1 -19950.753,E2 -19950.753} C_VEL
LIN {X 0,Y 254.971,Z 722.03,A -85,B 0,C 180,E1 -19952.392,E2 -19952.392} C_VEL
LIN {X 0,Y 251.407,Z 717.441,A -85,B 0,C 180,E1 -19954.266,E2 -19954.266} C_VEL
LIN {X 0,Y 248.415,Z 713.763,A -85,B 0,C 180,E1 -19955.975,E2 -19955.975} C_VEL
LIN {X 0,Y 247.604,Z 712.642,A -85,B 0,C 180,E1 -19956.475,E2 -19956.475} C_VEL
LIN {X 0,Y 244.831,Z 709.862,A -85,B 0,C 180,E1 -19958.209,E2 -19958.209} C_VEL
LIN {X 0,Y 243.316,Z 707.426,A -85,B 0,C 180,E1 -19959.307,E2 -19959.307} C_VEL
LIN {X 0,Y 240.496,Z 705.031,A -85,B 0,C 180,E1 -19961.359,E2 -19961.359} C_VEL
LIN {X 0,Y 238.625,Z 701.84,A -85,B 0,C 180,E1 -19963.039,E2 -19963.039} C_VEL
LIN {X 0,Y 235.699,Z 699.793,A -85,B 0,C 180,E1 -19965.759,E2 -19965.759} C_VEL
LIN {X 0,Y 233.39,Z 696.027,A -85,B 0,C 180,E1 -19968.712,E2 -19968.712} C_VEL
LIN {X 0,Y 229.349,Z 692.469,A -85,B 0,C 180,E1 -19977.804,E2 -19977.804} C_VEL
LIN {X 0,Y 229.217,Z 691.926,A -85,B 0,C 180,E1 -19980,E2 -19980} C_VEL
LIN {X 0,Y 229.338,Z 692.603,A -85,B 0,C 180,E1 -19982.634,E2 -19982.634} C_VEL
LIN {X 0,Y 233.642,Z 696.358,A -85,B 0,C 180,E1 -19992.045,E2 -19992.045} C_VEL
LIN {X 0,Y 235.826,Z 699.927,A -85,B 0,C 180,E1 -19994.783,E2 -19994.783} C_VEL
LIN {X 0,Y 238.948,Z 702.238,A -85,B 0,C 180,E1 -19997.656,E2 -19997.656} C_VEL
LIN {X 0,Y 240.789,Z 705.347,A -85,B 0,C 180,E1 -19999.279,E2 -19999.279} C_VEL
LIN {X 0,Y 243.629,Z 707.817,A -85,B 0,C 180,E1 -20001.324,E2 -20001.324} C_VEL
LIN {X 0,Y 245.997,Z 711.248,A -85,B 0,C 180,E1 -20002.963,E2 -20002.963} C_VEL
LIN {X 0,Y 248.128,Z 713.238,A -85,B 0,C 180,E1 -20004.248,E2 -20004.248} C_VEL
LIN {X 0,Y 250.902,Z 716.944,A -85,B 0,C 180,E1 -20005.872,E2 -20005.872} C_VEL
LIN {X 0,Y 252.23,Z 718.443,A -85,B 0,C 180,E1 -20006.586,E2 -20006.586} C_VEL
LIN {X 0,Y 255.357,Z 722.419,A -85,B 0,C 180,E1 -20008.202,E2 -20008.202} C_VEL
LIN {X 0,Y 260.508,Z 729.367,A -85,B 0,C 180,E1 -20010.636,E2 -20010.636} C_VEL
LIN {X 0,Y 265.205,Z 735.716,A -85,B 0,C 180,E1 -20012.637,E2 -20012.637} C_VEL
LIN {X 0,Y 276.111,Z 750.528,A -85,B 0,C 180,E1 -20016.681,E2 -20016.681} C_VEL
LIN {X 0,Y 283.679,Z 758.722,A -85,B 0,C 180,E1 -20019.026,E2 -20019.026} C_VEL
LIN {X 0,Y 291.15,Z 765.751,A -85,B 0,C 180,E1 -20021.093,E2 -20021.093} C_VEL
LIN {X 0,Y 298.749,Z 772.509,A -85,B 0,C 180,E1 -20023.235,E2 -20023.235} C_VEL
LIN {X 0,Y 306.175,Z 779.078,A -85,B 0,C 180,E1 -20025.505,E2 -20025.505} C_VEL
LIN {X 0,Y 313.211,Z 785.511,A -85,B 0,C 180,E1 -20027.896,E2 -20027.896} C_VEL
LIN {X 0,Y 316.906,Z 788.984,A -85,B 0,C 180,E1 -20029.271,E2 -20029.271} C_VEL
LIN {X 0,Y 324.192,Z 795.677,A -85,B 0,C 180,E1 -20032.087,E2 -20032.087} C_VEL
LIN {X 0,Y 329.374,Z 800.219,A -85,B 0,C 180,E1 -20034.175,E2 -20034.175} C_VEL
LIN {X 0,Y 335.835,Z 806.052,A -85,B 0,C 180,E1 -20036.915,E2 -20036.915} C_VEL
LIN {X 0,Y 339.466,Z 809.109,A -85,B 0,C 180,E1 -20038.522,E2 -20038.522} C_VEL
LIN {X 0,Y 343.995,Z 813.248,A -85,B 0,C 180,E1 -20040.638,E2 -20040.638} C_VEL
LIN {X 0,Y 347.524,Z 815.988,A -85,B 0,C 180,E1 -20042.349,E2 -20042.349} C_VEL
LIN {X 0,Y 351.48,Z 819.683,A -85,B 0,C 180,E1 -20044.421,E2 -20044.421} C_VEL
LIN {X 0,Y 355.848,Z 822.713,A -85,B 0,C 180,E1 -20046.81,E2 -20046.81} C_VEL
LIN {X 0,Y 359.317,Z 826.088,A -85,B 0,C 180,E1 -20048.976,E2 -20048.976} C_VEL
LIN {X 0,Y 363.104,Z 828.988,A -85,B 0,C 180,E1 -20051.514,E2 -20051.514} C_VEL
LIN {X 0,Y 365.897,Z 830.69,A -85,B 0,C 180,E1 -20053.565,E2 -20053.565} C_VEL
LIN {X 0,Y 368.55,Z 833.511,A -85,B 0,C 180,E1 -20055.917,E2 -20055.917} C_VEL
LIN {X 0,Y 370.822,Z 835.355,A -85,B 0,C 180,E1 -20058.206,E2 -20058.206} C_VEL
LIN {X 0,Y 372.948,Z 836.595,A -85,B 0,C 180,E1 -20060.765,E2 -20060.765} C_VEL
LIN {X 0,Y 374.74,Z 837.363,A -85,B 0,C 180,E1 -20063.539,E2 -20063.539} C_VEL
LIN {X 0,Y 375.627,Z 837.974,A -85,B 0,C 180,E1 -20065.708,E2 -20065.708} C_VEL
LIN {X 0,Y 376.209,Z 838.183,A -85,B 0,C 180,E1 -20067.859,E2 -20067.859} C_VEL
LIN {X 0,Y 376.418,Z 838.282,A -85,B 0,C 180,E1 -20070,E2 -20070} C_VEL
LIN {X 0,Y 376.209,Z 838.182,A -85,B 0,C 180,E1 -20072.141,E2 -20072.141} C_VEL
LIN {X 0,Y 375.485,Z 837.851,A -85,B 0,C 180,E1 -20074.748,E2 -20074.748} C_VEL
LIN {X 0,Y 374.418,Z 837.315,A -85,B 0,C 180,E1 -20077,E2 -20077} C_VEL
LIN {X 0,Y 372.552,Z 836.428,A -85,B 0,C 180,E1 -20079.775,E2 -20079.775} C_VEL
LIN {X 0,Y 370.453,Z 835.086,A -85,B 0,C 180,E1 -20082.176,E2 -20082.176} C_VEL
LIN {X 0,Y 367.783,Z 832.803,A -85,B 0,C 180,E1 -20084.796,E2 -20084.796} C_VEL
LIN {X 0,Y 365.187,Z 830.111,A -85,B 0,C 180,E1 -20086.984,E2 -20086.984} C_VEL
LIN {X 0,Y 361.799,Z 828.067,A -85,B 0,C 180,E1 -20089.395,E2 -20089.395} C_VEL
LIN {X 0,Y 358.086,Z 824.937,A -85,B 0,C 180,E1 -20091.823,E2 -20091.823} C_VEL
LIN {X 0,Y 355.522,Z 822.491,A -85,B 0,C 180,E1 -20093.372,E2 -20093.372} C_VEL
LIN {X 0,Y 350.977,Z 819.292,A -85,B 0,C 180,E1 -20095.855,E2 -20095.855} C_VEL
LIN {X 0,Y 346.126,Z 814.76,A -85,B 0,C 180,E1 -20098.352,E2 -20098.352} C_VEL
LIN {X 0,Y 341.622,Z 811.202,A -85,B 0,C 180,E1 -20100.477,E2 -20100.477} C_VEL
LIN {X 0,Y 337.347,Z 807.234,A -85,B 0,C 180,E1 -20102.437,E2 -20102.437} C_VEL
LIN {X 0,Y 332.234,Z 802.81,A -85,B 0,C 180,E1 -20104.635,E2 -20104.635} C_VEL
LIN {X 0,Y 328.758,Z 799.729,A -85,B 0,C 180,E1 -20106.076,E2 -20106.076} C_VEL
LIN {X 0,Y 323.413,Z 794.879,A -85,B 0,C 180,E1 -20108.225,E2 -20108.225} C_VEL
LIN {X 0,Y 316.72,Z 788.785,A -85,B 0,C 180,E1 -20110.801,E2 -20110.801} C_VEL
LIN {X 0,Y 312.672,Z 785.045,A -85,B 0,C 180,E1 -20112.291,E2 -20112.291} C_VEL
LIN {X 0,Y 305.887,Z 778.831,A -85,B 0,C 180,E1 -20114.583,E2 -20114.583} C_VEL
LIN {X 0,Y 300.508,Z 773.907,A -85,B 0,C 180,E1 -20116.247,E2 -20116.247} C_VEL
LIN {X 0,Y 294.743,Z 769.037,A -85,B 0,C 180,E1 -20117.908,E2 -20117.908} C_VEL
LIN {X 0,Y 288.361,Z 763.369,A -85,B 0,C 180,E1 -20119.656,E2 -20119.656} C_VEL
LIN {X 0,Y 278.237,Z 752.932,A -85,B 0,C 180,E1 -20122.631,E2 -20122.631} C_VEL
LIN {X 0,Y 272.179,Z 745.511,A -85,B 0,C 180,E1 -20124.679,E2 -20124.679} C_VEL
LIN {X 0,Y 261.983,Z 731.206,A -85,B 0,C 180,E1 -20128.724,E2 -20128.724} C_VEL
LIN {X 0,Y 257.969,Z 726.047,A -85,B 0,C 180,E1 -20130.523,E2 -20130.523} C_VEL
LIN {X 0,Y 254.853,Z 721.877,A -85,B 0,C 180,E1 -20132.044,E2 -20132.044} C_VEL
LIN {X 0,Y 251.983,Z 718.009,A -85,B 0,C 180,E1 -20133.555,E2 -20133.555} C_VEL
LIN {X 0,Y 248.62,Z 714.073,A -85,B 0,C 180,E1 -20135.442,E2 -20135.442} C_VEL
LIN {X 0,Y 247.66,Z 712.655,A -85,B 0,C 180,E1 -20136.037,E2 -20136.037} C_VEL
LIN {X 0,Y 244.82,Z 709.827,A -85,B 0,C 180,E1 -20137.811,E2 -20137.811} C_VEL
LIN {X 0,Y 243.359,Z 707.416,A -85,B 0,C 180,E1 -20138.874,E2 -20138.874} C_VEL
LIN {X 0,Y 240.664,Z 705.189,A -85,B 0,C 180,E1 -20140.821,E2 -20140.821} C_VEL
LIN {X 0,Y 238.896,Z 702.128,A -85,B 0,C 180,E1 -20142.395,E2 -20142.395} C_VEL
LIN {X 0,Y 235.348,Z 699.386,A -85,B 0,C 180,E1 -20145.738,E2 -20145.738} C_VEL
LIN {X 0,Y 233.562,Z 696.281,A -85,B 0,C 180,E1 -20148.061,E2 -20148.061} C_VEL
LIN {X 0,Y 230.041,Z 693.804,A -85,B 0,C 180,E1 -20154.302,E2 -20154.302} C_VEL
LIN {X 0,Y 229.217,Z 692.036,A -85,B 0,C 180,E1 -20159.122,E2 -20159.122} C_VEL
LIN {X 0,Y 229.307,Z 692.271,A -85,B 0,C 180,E1 -20161.757,E2 -20161.757} C_VEL
LIN {X 0,Y 230.544,Z 694.185,A -85,B 0,C 180,E1 -20166.565,E2 -20166.565} C_VEL
LIN {X 0,Y 233.701,Z 696.405,A -85,B 0,C 180,E1 -20171.712,E2 -20171.712} C_VEL
LIN {X 0,Y 235.795,Z 699.91,A -85,B 0,C 180,E1 -20174.345,E2 -20174.345} C_VEL
LIN {X 0,Y 238.91,Z 702.22,A -85,B 0,C 180,E1 -20177.218,E2 -20177.218} C_VEL
LIN {X 0,Y 240.745,Z 705.339,A -85,B 0,C 180,E1 -20178.841,E2 -20178.841} C_VEL
LIN {X 0,Y 243.657,Z 707.883,A -85,B 0,C 180,E1 -20180.939,E2 -20180.939} C_VEL
LIN {X 0,Y 245.682,Z 710.935,A -85,B 0,C 180,E1 -20182.357,E2 -20182.357} C_VEL
LIN {X 0,Y 248.189,Z 713.371,A -85,B 0,C 180,E1 -20183.882,E2 -20183.882} C_VEL
LIN {X 0,Y 251.052,Z 717.103,A -85,B 0,C 180,E1 -20185.546,E2 -20185.546} C_VEL
LIN {X 0,Y 252.332,Z 718.59,A -85,B 0,C 180,E1 -20186.235,E2 -20186.235} C_VEL
LIN {X 0,Y 256.459,Z 724.016,A -85,B 0,C 180,E1 -20188.346,E2 -20188.346} C_VEL
LIN {X 0,Y 260.395,Z 729.211,A -85,B 0,C 180,E1 -20190.178,E2 -20190.178} C_VEL
LIN {X 0,Y 265.104,Z 736.718,A -85,B 0,C 180,E1 -20192.245,E2 -20192.245} C_VEL
LIN {X 0,Y 272.262,Z 749.346,A -85,B 0,C 180,E1 -20195.111,E2 -20195.111} C_VEL
LIN {X 0,Y 278.697,Z 762.205,A -85,B 0,C 180,E1 -20197.472,E2 -20197.472} C_VEL
LIN {X 0,Y 284.288,Z 774.383,A -85,B 0,C 180,E1 -20199.383,E2 -20199.383} C_VEL
LIN {X 0,Y 286.407,Z 779.676,A -85,B 0,C 180,E1 -20200.094,E2 -20200.094} C_VEL
LIN {X 0,Y 281.985,Z 851.539,A -85,B 0,C 180,E1 -20201.778,E2 -20201.778} C_VEL
LIN {X 0,Y 281.205,Z 857.39,A -85,B 0,C 180,E1 -20201.817,E2 -20201.817} C_VEL
LIN {X 0,Y 276.219,Z 876.48,A -85,B 0,C 180,E1 -20201.386,E2 -20201.386} C_VEL
LIN {X 0,Y 275.365,Z 882.329,A -85,B 0,C 180,E1 -20201.423,E2 -20201.423} C_VEL
LIN {X 0,Y 273.784,Z 899.312,A -85,B 0,C 180,E1 -20201.943,E2 -20201.943} C_VEL
LIN {X 0,Y 271.65,Z 913.565,A -85,B 0,C 180,E1 -20202.537,E2 -20202.537} C_VEL
LIN {X 0,Y 268.991,Z 926.982,A -85,B 0,C 180,E1 -20203.258,E2 -20203.258} C_VEL
LIN {X 0,Y 266.458,Z 938.366,A -85,B 0,C 180,E1 -20204.051,E2 -20204.051} C_VEL
LIN {X 0,Y 262.969,Z 951.597,A -85,B 0,C 180,E1 -20205.181,E2 -20205.181} C_VEL
LIN {X 0,Y 259.035,Z 964.326,A -85,B 0,C 180,E1 -20206.493,E2 -20206.493} C_VEL
LIN {X 0,Y 255.194,Z 975.805,A -85,B 0,C 180,E1 -20207.939,E2 -20207.939} C_VEL
LIN {X 0,Y 251.412,Z 986.2,A -85,B 0,C 180,E1 -20209.485,E2 -20209.485} C_VEL
LIN {X 0,Y 247.129,Z 996.605,A -85,B 0,C 180,E1 -20211.271,E2 -20211.271} C_VEL
LIN {X 0,Y 243.256,Z 1005.873,A -85,B 0,C 180,E1 -20213.167,E2 -20213.167} C_VEL
LIN {X 0,Y 239.086,Z 1015.184,A -85,B 0,C 180,E1 -20215.393,E2 -20215.393} C_VEL
LIN {X 0,Y 235.017,Z 1024.126,A -85,B 0,C 180,E1 -20217.941,E2 -20217.941} C_VEL
LIN {X 0,Y 230.959,Z 1032.726,A -85,B 0,C 180,E1 -20220.866,E2 -20220.866} C_VEL
LIN {X 0,Y 227.799,Z 1039.53,A -85,B 0,C 180,E1 -20223.619,E2 -20223.619} C_VEL
LIN {X 0,Y 224.699,Z 1046.425,A -85,B 0,C 180,E1 -20226.986,E2 -20226.986} C_VEL
LIN {X 0,Y 222.675,Z 1051.079,A -85,B 0,C 180,E1 -20229.686,E2 -20229.686} C_VEL
LIN {X 0,Y 220.723,Z 1056.187,A -85,B 0,C 180,E1 -20233.348,E2 -20233.348} C_VEL
LIN {X 0,Y 219.375,Z 1060.195,A -85,B 0,C 180,E1 -20237.041,E2 -20237.041} C_VEL
LIN {X 0,Y 218.703,Z 1063.163,A -85,B 0,C 180,E1 -20240.754,E2 -20240.754} C_VEL
LIN {X 0,Y 218.542,Z 1064.355,A -85,B 0,C 180,E1 -20242.61,E2 -20242.61} C_VEL
LIN {X 0,Y 218.45,Z 1065.835,A -85,B 0,C 180,E1 -20246.311,E2 -20246.311} C_VEL
LIN {X 0,Y 218.628,Z 1066.331,A -85,B 0,C 180,E1 -20250,E2 -20250} C_VEL
LIN {X 0,Y 218.481,Z 1065.608,A -85,B 0,C 180,E1 -20254.292,E2 -20254.292} C_VEL
LIN {X 0,Y 218.542,Z 1064.355,A -85,B 0,C 180,E1 -20257.39,E2 -20257.39} C_VEL
LIN {X 0,Y 218.966,Z 1061.875,A -85,B 0,C 180,E1 -20261.103,E2 -20261.103} C_VEL
LIN {X 0,Y 220.337,Z 1057.277,A -85,B 0,C 180,E1 -20265.731,E2 -20265.731} C_VEL
LIN {X 0,Y 221.619,Z 1053.781,A -85,B 0,C 180,E1 -20268.488,E2 -20268.488} C_VEL
LIN {X 0,Y 223.959,Z 1048.047,A -85,B 0,C 180,E1 -20272.121,E2 -20272.121} C_VEL
LIN {X 0,Y 226.257,Z 1042.984,A -85,B 0,C 180,E1 -20274.792,E2 -20274.792} C_VEL
LIN {X 0,Y 229.897,Z 1034.948,A -85,B 0,C 180,E1 -20278.283,E2 -20278.283} C_VEL
LIN {X 0,Y 233.209,Z 1027.965,A -85,B 0,C 180,E1 -20280.817,E2 -20280.817} C_VEL
LIN {X 0,Y 236.945,Z 1019.999,A -85,B 0,C 180,E1 -20283.279,E2 -20283.279} C_VEL
LIN {X 0,Y 241.048,Z 1010.888,A -85,B 0,C 180,E1 -20285.669,E2 -20285.669} C_VEL
LIN {X 0,Y 244.79,Z 1002.323,A -85,B 0,C 180,E1 -20287.595,E2 -20287.595} C_VEL
LIN {X 0,Y 249.161,Z 991.548,A -85,B 0,C 180,E1 -20289.655,E2 -20289.655} C_VEL
LIN {X 0,Y 253.515,Z 980.384,A -85,B 0,C 180,E1 -20291.424,E2 -20291.424} C_VEL
LIN {X 0,Y 257.673,Z 968.64,A -85,B 0,C 180,E1 -20292.989,E2 -20292.989} C_VEL
LIN {X 0,Y 261.486,Z 956.621,A -85,B 0,C 180,E1 -20294.33,E2 -20294.33} C_VEL
LIN {X 0,Y 264.953,Z 944.307,A -85,B 0,C 180,E1 -20295.467,E2 -20295.467} C_VEL
LIN {X 0,Y 267.952,Z 931.766,A -85,B 0,C 180,E1 -20296.431,E2 -20296.431} C_VEL
LIN {X 0,Y 270.649,Z 918.841,A -85,B 0,C 180,E1 -20297.208,E2 -20297.208} C_VEL
LIN {X 0,Y 272.917,Z 905.428,A -85,B 0,C 180,E1 -20297.829,E2 -20297.829} C_VEL
LIN {X 0,Y 274.582,Z 892.297,A -85,B 0,C 180,E1 -20298.281,E2 -20298.281} C_VEL
LIN {X 0,Y 276.442,Z 864.787,A -85,B 0,C 180,E1 -20299.001,E2 -20299.001} C_VEL
LIN {X 0,Y 281.714,Z 782.01,A -85,B 0,C 180,E1 -20300.952,E2 -20300.952} C_VEL
LIN {X 0,Y 276.261,Z 769.455,A -85,B 0,C 180,E1 -20302.882,E2 -20302.882} C_VEL
LIN {X 0,Y 269.311,Z 755.184,A -85,B 0,C 180,E1 -20305.517,E2 -20305.517} C_VEL
LIN {X 0,Y 262.684,Z 743.084,A -85,B 0,C 180,E1 -20308.271,E2 -20308.271} C_VEL
LIN {X 0,Y 257.887,Z 735.197,A -85,B 0,C 180,E1 -20310.456,E2 -20310.456} C_VEL
LIN {X 0,Y 252.912,Z 728.447,A -85,B 0,C 180,E1 -20312.898,E2 -20312.898} C_VEL
LIN {X 0,Y 249.278,Z 723.71,A -85,B 0,C 180,E1 -20314.874,E2 -20314.874} C_VEL
LIN {X 0,Y 246.267,Z 719.821,A -85,B 0,C 180,E1 -20316.673,E2 -20316.673} C_VEL
LIN {X 0,Y 242.635,Z 715.711,A -85,B 0,C 180,E1 -20319.056,E2 -20319.056} C_VEL
LIN {X 0,Y 241.658,Z 714.106,A -85,B 0,C 180,E1 -20319.796,E2 -20319.796} C_VEL
LIN {X 0,Y 239.014,Z 711.736,A -85,B 0,C 180,E1 -20321.795,E2 -20321.795} C_VEL
LIN {X 0,Y 237.236,Z 708.674,A -85,B 0,C 180,E1 -20323.444,E2 -20323.444} C_VEL
LIN {X 0,Y 234.36,Z 706.507,A -85,B 0,C 180,E1 -20326.229,E2 -20326.229} C_VEL
LIN {X 0,Y 232.374,Z 703.019,A -85,B 0,C 180,E1 -20328.883,E2 -20328.883} C_VEL
LIN {X 0,Y 228.374,Z 699.108,A -85,B 0,C 180,E1 -20339.118,E2 -20339.118} C_VEL
LIN {X 0,Y 228.397,Z 699.276,A -85,B 0,C 180,E1 -20341.763,E2 -20341.763} C_VEL
LIN {X 0,Y 232.505,Z 703.229,A -85,B 0,C 180,E1 -20351.717,E2 -20351.717} C_VEL
LIN {X 0,Y 234.483,Z 706.654,A -85,B 0,C 180,E1 -20354.316,E2 -20354.316} C_VEL
LIN {X 0,Y 237.419,Z 708.91,A -85,B 0,C 180,E1 -20357.133,E2 -20357.133} C_VEL
LIN {X 0,Y 239.424,Z 712.202,A -85,B 0,C 180,E1 -20358.948,E2 -20358.948} C_VEL
LIN {X 0,Y 241.954,Z 714.45,A -85,B 0,C 180,E1 -20360.826,E2 -20360.826} C_VEL
LIN {X 0,Y 244.322,Z 717.865,A -85,B 0,C 180,E1 -20362.515,E2 -20362.515} C_VEL
LIN {X 0,Y 246.323,Z 719.853,A -85,B 0,C 180,E1 -20363.766,E2 -20363.766} C_VEL
LIN {X 0,Y 249.165,Z 723.607,A -85,B 0,C 180,E1 -20365.472,E2 -20365.472} C_VEL
LIN {X 0,Y 250.605,Z 725.498,A -85,B 0,C 180,E1 -20366.282,E2 -20366.282} C_VEL
LIN {X 0,Y 254.063,Z 730.032,A -85,B 0,C 180,E1 -20368.102,E2 -20368.102} C_VEL
LIN {X 0,Y 259.994,Z 737.995,A -85,B 0,C 180,E1 -20370.903,E2 -20370.903} C_VEL
LIN {X 0,Y 273.776,Z 757.06,A -85,B 0,C 180,E1 -20376.3,E2 -20376.3} C_VEL
LIN {X 0,Y 281.108,Z 765.038,A -85,B 0,C 180,E1 -20378.625,E2 -20378.625} C_VEL
LIN {X 0,Y 288.146,Z 771.76,A -85,B 0,C 180,E1 -20380.61,E2 -20380.61} C_VEL
LIN {X 0,Y 296.298,Z 778.879,A -85,B 0,C 180,E1 -20382.854,E2 -20382.854} C_VEL
LIN {X 0,Y 303.617,Z 785.317,A -85,B 0,C 180,E1 -20385.065,E2 -20385.065} C_VEL
LIN {X 0,Y 308.415,Z 789.597,A -85,B 0,C 180,E1 -20386.62,E2 -20386.62} C_VEL
LIN {X 0,Y 314.465,Z 795.047,A -85,B 0,C 180,E1 -20388.744,E2 -20388.744} C_VEL
LIN {X 0,Y 319.952,Z 799.978,A -85,B 0,C 180,E1 -20390.817,E2 -20390.817} C_VEL
LIN {X 0,Y 326.566,Z 806.068,A -85,B 0,C 180,E1 -20393.438,E2 -20393.438} C_VEL
LIN {X 0,Y 330.197,Z 809.152,A -85,B 0,C 180,E1 -20394.924,E2 -20394.924} C_VEL
LIN {X 0,Y 335.234,Z 813.565,A -85,B 0,C 180,E1 -20397.073,E2 -20397.073} C_VEL
LIN {X 0,Y 338.251,Z 816.222,A -85,B 0,C 180,E1 -20398.415,E2 -20398.415} C_VEL
LIN {X 0,Y 342.981,Z 820.369,A -85,B 0,C 180,E1 -20400.605,E2 -20400.605} C_VEL
LIN {X 0,Y 346.097,Z 822.793,A -85,B 0,C 180,E1 -20402.109,E2 -20402.109} C_VEL
LIN {X 0,Y 350.307,Z 826.643,A -85,B 0,C 180,E1 -20404.285,E2 -20404.285} C_VEL
LIN {X 0,Y 354.648,Z 829.643,A -85,B 0,C 180,E1 -20406.651,E2 -20406.651} C_VEL
LIN {X 0,Y 358.082,Z 832.962,A -85,B 0,C 180,E1 -20408.772,E2 -20408.772} C_VEL
LIN {X 0,Y 361.927,Z 835.891,A -85,B 0,C 180,E1 -20411.312,E2 -20411.312} C_VEL
LIN {X 0,Y 364.837,Z 837.68,A -85,B 0,C 180,E1 -20413.442,E2 -20413.442} C_VEL
LIN {X 0,Y 367.627,Z 840.574,A -85,B 0,C 180,E1 -20415.88,E2 -20415.88} C_VEL
LIN {X 0,Y 369.915,Z 842.397,A -85,B 0,C 180,E1 -20418.177,E2 -20418.177} C_VEL
LIN {X 0,Y 372.063,Z 843.613,A -85,B 0,C 180,E1 -20420.743,E2 -20420.743} C_VEL
LIN {X 0,Y 373.868,Z 844.382,A -85,B 0,C 180,E1 -20423.524,E2 -20423.524} C_VEL
LIN {X 0,Y 374.757,Z 845.014,A -85,B 0,C 180,E1 -20425.698,E2 -20425.698} C_VEL
LIN {X 0,Y 375.344,Z 845.201,A -85,B 0,C 180,E1 -20427.854,E2 -20427.854} C_VEL
LIN {X 0,Y 375.553,Z 845.328,A -85,B 0,C 180,E1 -20430,E2 -20430} C_VEL
LIN {X 0,Y 375.343,Z 845.201,A -85,B 0,C 180,E1 -20432.146,E2 -20432.146} C_VEL
LIN {X 0,Y 374.615,Z 844.898,A -85,B 0,C 180,E1 -20434.759,E2 -20434.759} C_VEL
LIN {X 0,Y 373.871,Z 844.359,A -85,B 0,C 180,E1 -20436.476,E2 -20436.476} C_VEL
LIN {X 0,Y 372.496,Z 843.747,A -85,B 0,C 180,E1 -20438.681,E2 -20438.681} C_VEL
LIN {X 0,Y 370.71,Z 842.937,A -85,B 0,C 180,E1 -20440.928,E2 -20440.928} C_VEL
LIN {X 0,Y 368.16,Z 841.038,A -85,B 0,C 180,E1 -20443.607,E2 -20443.607} C_VEL
LIN {X 0,Y 365.668,Z 838.616,A -85,B 0,C 180,E1 -20445.872,E2 -20445.872} C_VEL
LIN {X 0,Y 364.036,Z 837.05,A -85,B 0,C 180,E1 -20447.186,E2 -20447.186} C_VEL
LIN {X 0,Y 360.623,Z 834.967,A -85,B 0,C 180,E1 -20449.574,E2 -20449.574} C_VEL
LIN {X 0,Y 356.925,Z 831.912,A -85,B 0,C 180,E1 -20451.969,E2 -20451.969} C_VEL
LIN {X 0,Y 354.297,Z 829.395,A -85,B 0,C 180,E1 -20453.543,E2 -20453.543} C_VEL
LIN {X 0,Y 349.774,Z 826.244,A -85,B 0,C 180,E1 -20455.996,E2 -20455.996} C_VEL
LIN {X 0,Y 344.485,Z 821.435,A -85,B 0,C 180,E1 -20458.688,E2 -20458.688} C_VEL
LIN {X 0,Y 339.982,Z 817.848,A -85,B 0,C 180,E1 -20460.797,E2 -20460.797} C_VEL
LIN {X 0,Y 335.62,Z 813.855,A -85,B 0,C 180,E1 -20462.761,E2 -20462.761} C_VEL
LIN {X 0,Y 330.467,Z 809.422,A -85,B 0,C 180,E1 -20464.962,E2 -20464.962} C_VEL
LIN {X 0,Y 327.669,Z 806.898,A -85,B 0,C 180,E1 -20466.117,E2 -20466.117} C_VEL
LIN {X 0,Y 322.121,Z 802.064,A -85,B 0,C 180,E1 -20468.328,E2 -20468.328} C_VEL
LIN {X 0,Y 314.802,Z 795.38,A -85,B 0,C 180,E1 -20471.126,E2 -20471.126} C_VEL
LIN {X 0,Y 309.002,Z 790.149,A -85,B 0,C 180,E1 -20473.186,E2 -20473.186} C_VEL
LIN {X 0,Y 303.787,Z 785.44,A -85,B 0,C 180,E1 -20474.881,E2 -20474.881} C_VEL
LIN {X 0,Y 298.352,Z 780.547,A -85,B 0,C 180,E1 -20476.543,E2 -20476.543} C_VEL
LIN {X 0,Y 291.41,Z 774.613,A -85,B 0,C 180,E1 -20478.512,E2 -20478.512} C_VEL
LIN {X 0,Y 282.585,Z 766.536,A -85,B 0,C 180,E1 -20480.94,E2 -20480.94} C_VEL
LIN {X 0,Y 275.181,Z 758.643,A -85,B 0,C 180,E1 -20483.232,E2 -20483.232} C_VEL
LIN {X 0,Y 266.997,Z 748.287,A -85,B 0,C 180,E1 -20486.16,E2 -20486.16} C_VEL
LIN {X 0,Y 260.478,Z 738.743,A -85,B 0,C 180,E1 -20488.879,E2 -20488.879} C_VEL
LIN {X 0,Y 255.704,Z 732.278,A -85,B 0,C 180,E1 -20491.082,E2 -20491.082} C_VEL
LIN {X 0,Y 252.473,Z 727.95,A -85,B 0,C 180,E1 -20492.715,E2 -20492.715} C_VEL
LIN {X 0,Y 249.168,Z 723.576,A -85,B 0,C 180,E1 -20494.529,E2 -20494.529} C_VEL
LIN {X 0,Y 246.245,Z 719.763,A -85,B 0,C 180,E1 -20496.282,E2 -20496.282} C_VEL
LIN {X 0,Y 242.715,Z 715.803,A -85,B 0,C 180,E1 -20498.592,E2 -20498.592} C_VEL
LIN {X 0,Y 241.604,Z 714.058,A -85,B 0,C 180,E1 -20499.428,E2 -20499.428} C_VEL
LIN {X 0,Y 238.936,Z 711.595,A -85,B 0,C 180,E1 -20501.456,E2 -20501.456} C_VEL
LIN {X 0,Y 237.16,Z 708.64,A -85,B 0,C 180,E1 -20503.101,E2 -20503.101} C_VEL
LIN {X 0,Y 234.296,Z 706.441,A -85,B 0,C 180,E1 -20505.894,E2 -20505.894} C_VEL
LIN {X 0,Y 232.387,Z 703.129,A -85,B 0,C 180,E1 -20508.443,E2 -20508.443} C_VEL
LIN {X 0,Y 228.351,Z 699.089,A -85,B 0,C 180,E1 -20519.119,E2 -20519.119} C_VEL
LIN {X 0,Y 228.399,Z 699.231,A -85,B 0,C 180,E1 -20521.323,E2 -20521.323} C_VEL
LIN {X 0,Y 232.597,Z 703.343,A -85,B 0,C 180,E1 -20531.437,E2 -20531.437} C_VEL
LIN {X 0,Y 234.547,Z 706.737,A -85,B 0,C 180,E1 -20533.981,E2 -20533.981} C_VEL
LIN {X 0,Y 237.402,Z 708.914,A -85,B 0,C 180,E1 -20536.713,E2 -20536.713} C_VEL
LIN {X 0,Y 239.257,Z 712.039,A -85,B 0,C 180,E1 -20538.408,E2 -20538.408} C_VEL
LIN {X 0,Y 241.989,Z 714.588,A -85,B 0,C 180,E1 -20540.453,E2 -20540.453} C_VEL
LIN {X 0,Y 244.417,Z 718.005,A -85,B 0,C 180,E1 -20542.173,E2 -20542.173} C_VEL
LIN {X 0,Y 246.345,Z 719.907,A -85,B 0,C 180,E1 -20543.374,E2 -20543.374} C_VEL
LIN {X 0,Y 249.275,Z 723.732,A -85,B 0,C 180,E1 -20545.127,E2 -20545.127} C_VEL
LIN {X 0,Y 254.106,Z 730.086,A -85,B 0,C 180,E1 -20547.716,E2 -20547.716} C_VEL
LIN {X 0,Y 257.887,Z 735.196,A -85,B 0,C 180,E1 -20549.544,E2 -20549.544} C_VEL
LIN {X 0,Y 262.581,Z 742.964,A -85,B 0,C 180,E1 -20551.686,E2 -20551.686} C_VEL
LIN {X 0,Y 269.402,Z 755.368,A -85,B 0,C 180,E1 -20554.52,E2 -20554.52} C_VEL
LIN {X 0,Y 275.423,Z 767.742,A -85,B 0,C 180,E1 -20556.816,E2 -20556.816} C_VEL
LIN {X 0,Y 280.358,Z 778.764,A -85,B 0,C 180,E1 -20558.577,E2 -20558.577} C_VEL
LIN {X 0,Y 281.713,Z 781.943,A -85,B 0,C 180,E1 -20559.045,E2 -20559.045} C_VEL
LIN {X 0,Y 275.365,Z 882.329,A -85,B 0,C 180,E1 -20561.423,E2 -20561.423} C_VEL
LIN {X 0,Y 274.493,Z 888.165,A -85,B 0,C 180,E1 -20561.478,E2 -20561.478} C_VEL
LIN {X 0,Y 271.752,Z 897.657,A -85,B 0,C 180,E1 -20561.347,E2 -20561.347} C_VEL
LIN {X 0,Y 269.182,Z 905.167,A -85,B 0,C 180,E1 -20561.253,E2 -20561.253} C_VEL
LIN {X 0,Y 267.48,Z 910.848,A -85,B 0,C 180,E1 -20561.314,E2 -20561.314} C_VEL
LIN {X 0,Y 267.028,Z 912.737,A -85,B 0,C 180,E1 -20561.385,E2 -20561.385} C_VEL
LIN {X 0,Y 264.171,Z 926.776,A -85,B 0,C 180,E1 -20562.135,E2 -20562.135} C_VEL
LIN {X 0,Y 261.556,Z 938.16,A -85,B 0,C 180,E1 -20562.93,E2 -20562.93} C_VEL
LIN {X 0,Y 257.962,Z 951.39,A -85,B 0,C 180,E1 -20564.065,E2 -20564.065} C_VEL
LIN {X 0,Y 253.916,Z 964.12,A -85,B 0,C 180,E1 -20565.387,E2 -20565.387} C_VEL
LIN {X 0,Y 249.926,Z 975.598,A -85,B 0,C 180,E1 -20566.84,E2 -20566.84} C_VEL
LIN {X 0,Y 245.949,Z 986.162,A -85,B 0,C 180,E1 -20568.431,E2 -20568.431} C_VEL
LIN {X 0,Y 241.565,Z 996.398,A -85,B 0,C 180,E1 -20570.205,E2 -20570.205} C_VEL
LIN {X 0,Y 237.536,Z 1005.665,A -85,B 0,C 180,E1 -20572.127,E2 -20572.127} C_VEL
LIN {X 0,Y 232.883,Z 1015.625,A -85,B 0,C 180,E1 -20574.569,E2 -20574.569} C_VEL
LIN {X 0,Y 228.966,Z 1023.918,A -85,B 0,C 180,E1 -20576.988,E2 -20576.988} C_VEL
LIN {X 0,Y 224.688,Z 1032.517,A -85,B 0,C 180,E1 -20579.97,E2 -20579.97} C_VEL
LIN {X 0,Y 221.416,Z 1039.172,A -85,B 0,C 180,E1 -20582.717,E2 -20582.717} C_VEL
LIN {X 0,Y 218.063,Z 1046.216,A -85,B 0,C 180,E1 -20586.243,E2 -20586.243} C_VEL
LIN {X 0,Y 215.922,Z 1050.871,A -85,B 0,C 180,E1 -20589.021,E2 -20589.021} C_VEL
LIN {X 0,Y 213.815,Z 1055.978,A -85,B 0,C 180,E1 -20592.793,E2 -20592.793} C_VEL
LIN {X 0,Y 212.399,Z 1059.987,A -85,B 0,C 180,E1 -20596.608,E2 -20596.608} C_VEL
LIN {X 0,Y 211.63,Z 1062.956,A -85,B 0,C 180,E1 -20600.442,E2 -20600.442} C_VEL
LIN {X 0,Y 211.451,Z 1064.149,A -85,B 0,C 180,E1 -20602.36,E2 -20602.36} C_VEL
LIN {X 0,Y 211.357,Z 1065.629,A -85,B 0,C 180,E1 -20606.187,E2 -20606.187} C_VEL
LIN {X 0,Y 211.545,Z 1066.126,A -85,B 0,C 180,E1 -20610,E2 -20610} C_VEL
LIN {X 0,Y 211.367,Z 1065.546,A -85,B 0,C 180,E1 -20614.047,E2 -20614.047} C_VEL
LIN {X 0,Y 211.451,Z 1064.149,A -85,B 0,C 180,E1 -20617.64,E2 -20617.64} C_VEL
LIN {X 0,Y 211.923,Z 1061.667,A -85,B 0,C 180,E1 -20621.477,E2 -20621.477} C_VEL
LIN {X 0,Y 213.429,Z 1057.069,A -85,B 0,C 180,E1 -20626.254,E2 -20626.254} C_VEL
LIN {X 0,Y 215.339,Z 1052.222,A -85,B 0,C 180,E1 -20630.04,E2 -20630.04} C_VEL
LIN {X 0,Y 217.295,Z 1047.838,A -85,B 0,C 180,E1 -20632.837,E2 -20632.837} C_VEL
LIN {X 0,Y 219.724,Z 1042.775,A -85,B 0,C 180,E1 -20635.581,E2 -20635.581} C_VEL
LIN {X 0,Y 223.593,Z 1034.74,A -85,B 0,C 180,E1 -20639.156,E2 -20639.156} C_VEL
LIN {X 0,Y 227.042,Z 1027.756,A -85,B 0,C 180,E1 -20641.75,E2 -20641.75} C_VEL
LIN {X 0,Y 230.947,Z 1019.79,A -85,B 0,C 180,E1 -20644.261,E2 -20644.261} C_VEL
LIN {X 0,Y 235.248,Z 1010.68,A -85,B 0,C 180,E1 -20646.69,E2 -20646.69} C_VEL
LIN {X 0,Y 239.112,Z 1002.114,A -85,B 0,C 180,E1 -20648.65,E2 -20648.65} C_VEL
LIN {X 0,Y 243.717,Z 991.342,A -85,B 0,C 180,E1 -20650.724,E2 -20650.724} C_VEL
LIN {X 0,Y 248.184,Z 980.177,A -85,B 0,C 180,E1 -20652.519,E2 -20652.519} C_VEL
LIN {X 0,Y 252.483,Z 968.433,A -85,B 0,C 180,E1 -20654.097,E2 -20654.097} C_VEL
LIN {X 0,Y 256.436,Z 956.414,A -85,B 0,C 180,E1 -20655.443,E2 -20655.443} C_VEL
LIN {X 0,Y 260.006,Z 944.101,A -85,B 0,C 180,E1 -20656.587,E2 -20656.587} C_VEL
LIN {X 0,Y 263.097,Z 931.56,A -85,B 0,C 180,E1 -20657.554,E2 -20657.554} C_VEL
LIN {X 0,Y 265.968,Z 918.234,A -85,B 0,C 180,E1 -20658.347,E2 -20658.347} C_VEL
LIN {X 0,Y 268.276,Z 904.747,A -85,B 0,C 180,E1 -20658.969,E2 -20658.969} C_VEL
LIN {X 0,Y 269.91,Z 891.951,A -85,B 0,C 180,E1 -20659.413,E2 -20659.413} C_VEL
LIN {X 0,Y 271.85,Z 864.384,A -85,B 0,C 180,E1 -20660.135,E2 -20660.135} C_VEL
LIN {X 0,Y 277.068,Z 784.542,A -85,B 0,C 180,E1 -20662.039,E2 -20662.039} C_VEL
LIN {X 0,Y 271.553,Z 771.83,A -85,B 0,C 180,E1 -20664.101,E2 -20664.101} C_VEL
LIN {X 0,Y 265.636,Z 759.51,A -85,B 0,C 180,E1 -20666.472,E2 -20666.472} C_VEL
LIN {X 0,Y 259.041,Z 747.279,A -85,B 0,C 180,E1 -20669.366,E2 -20669.366} C_VEL
LIN {X 0,Y 255.043,Z 740.644,A -85,B 0,C 180,E1 -20671.281,E2 -20671.281} C_VEL
LIN {X 0,Y 250.311,Z 734.192,A -85,B 0,C 180,E1 -20673.71,E2 -20673.71} C_VEL
LIN {X 0,Y 247.077,Z 729.855,A -85,B 0,C 180,E1 -20675.552,E2 -20675.552} C_VEL
LIN {X 0,Y 243.726,Z 725.557,A -85,B 0,C 180,E1 -20677.649,E2 -20677.649} C_VEL
LIN {X 0,Y 240.818,Z 722.071,A -85,B 0,C 180,E1 -20679.667,E2 -20679.667} C_VEL
LIN {X 0,Y 239.844,Z 720.666,A -85,B 0,C 180,E1 -20680.418,E2 -20680.418} C_VEL
LIN {X 0,Y 237.2,Z 717.942,A -85,B 0,C 180,E1 -20682.542,E2 -20682.542} C_VEL
LIN {X 0,Y 235.671,Z 715.414,A -85,B 0,C 180,E1 -20684.019,E2 -20684.019} C_VEL
LIN {X 0,Y 232.774,Z 712.885,A -85,B 0,C 180,E1 -20687.023,E2 -20687.023} C_VEL
LIN {X 0,Y 231.208,Z 709.874,A -85,B 0,C 180,E1 -20689.27,E2 -20689.27} C_VEL
LIN {X 0,Y 227.511,Z 706.139,A -85,B 0,C 180,E1 -20699.115,E2 -20699.115} C_VEL
LIN {X 0,Y 227.527,Z 706.365,A -85,B 0,C 180,E1 -20701.77,E2 -20701.77} C_VEL
LIN {X 0,Y 231.445,Z 710.243,A -85,B 0,C 180,E1 -20711.494,E2 -20711.494} C_VEL
LIN {X 0,Y 233.155,Z 713.377,A -85,B 0,C 180,E1 -20713.842,E2 -20713.842} C_VEL
LIN {X 0,Y 236.032,Z 715.794,A -85,B 0,C 180,E1 -20716.728,E2 -20716.728} C_VEL
LIN {X 0,Y 238.196,Z 719.154,A -85,B 0,C 180,E1 -20718.715,E2 -20718.715} C_VEL
LIN {X 0,Y 240.356,Z 721.227,A -85,B 0,C 180,E1 -20720.373,E2 -20720.373} C_VEL
LIN {X 0,Y 243.027,Z 724.883,A -85,B 0,C 180,E1 -20722.306,E2 -20722.306} C_VEL
LIN {X 0,Y 244.606,Z 726.599,A -85,B 0,C 180,E1 -20723.325,E2 -20723.325} C_VEL
LIN {X 0,Y 247.662,Z 730.495,A -85,B 0,C 180,E1 -20725.192,E2 -20725.192} C_VEL
LIN {X 0,Y 252.556,Z 737.318,A -85,B 0,C 180,E1 -20727.889,E2 -20727.889} C_VEL
LIN {X 0,Y 255.945,Z 741.97,A -85,B 0,C 180,E1 -20729.564,E2 -20729.564} C_VEL
LIN {X 0,Y 260.391,Z 748.419,A -85,B 0,C 180,E1 -20731.594,E2 -20731.594} C_VEL
LIN {X 0,Y 270.938,Z 762.991,A -85,B 0,C 180,E1 -20735.735,E2 -20735.735} C_VEL
LIN {X 0,Y 278.323,Z 771.147,A -85,B 0,C 180,E1 -20738.148,E2 -20738.148} C_VEL
LIN {X 0,Y 285.612,Z 778.142,A -85,B 0,C 180,E1 -20740.254,E2 -20740.254} C_VEL
LIN {X 0,Y 293.471,Z 784.968,A -85,B 0,C 180,E1 -20742.399,E2 -20742.399} C_VEL
LIN {X 0,Y 300.745,Z 791.261,A -85,B 0,C 180,E1 -20744.511,E2 -20744.511} C_VEL
LIN {X 0,Y 306.848,Z 796.672,A -85,B 0,C 180,E1 -20746.466,E2 -20746.466} C_VEL
LIN {X 0,Y 312.403,Z 801.511,A -85,B 0,C 180,E1 -20748.374,E2 -20748.374} C_VEL
LIN {X 0,Y 317.967,Z 806.497,A -85,B 0,C 180,E1 -20750.45,E2 -20750.45} C_VEL
LIN {X 0,Y 324.621,Z 812.584,A -85,B 0,C 180,E1 -20753.066,E2 -20753.066} C_VEL
LIN {X 0,Y 328.58,Z 815.888,A -85,B 0,C 180,E1 -20754.661,E2 -20754.661} C_VEL
LIN {X 0,Y 333.612,Z 820.292,A -85,B 0,C 180,E1 -20756.79,E2 -20756.79} C_VEL
LIN {X 0,Y 336.753,Z 823.017,A -85,B 0,C 180,E1 -20758.175,E2 -20758.175} C_VEL
LIN {X 0,Y 341.646,Z 827.25,A -85,B 0,C 180,E1 -20760.417,E2 -20760.417} C_VEL
LIN {X 0,Y 344.624,Z 829.538,A -85,B 0,C 180,E1 -20761.844,E2 -20761.844} C_VEL
LIN {X 0,Y 348.95,Z 833.475,A -85,B 0,C 180,E1 -20764.058,E2 -20764.058} C_VEL
LIN {X 0,Y 354.106,Z 837.187,A -85,B 0,C 180,E1 -20766.871,E2 -20766.871} C_VEL
LIN {X 0,Y 357.536,Z 840.387,A -85,B 0,C 180,E1 -20769.001,E2 -20769.001} C_VEL
LIN {X 0,Y 361.385,Z 843.172,A -85,B 0,C 180,E1 -20771.562,E2 -20771.562} C_VEL
LIN {X 0,Y 363.722,Z 844.595,A -85,B 0,C 180,E1 -20773.271,E2 -20773.271} C_VEL
LIN {X 0,Y 366.408,Z 847.368,A -85,B 0,C 180,E1 -20775.561,E2 -20775.561} C_VEL
LIN {X 0,Y 368.767,Z 849.259,A -85,B 0,C 180,E1 -20777.899,E2 -20777.899} C_VEL
LIN {X 0,Y 370.822,Z 850.495,A -85,B 0,C 180,E1 -20780.237,E2 -20780.237} C_VEL
LIN {X 0,Y 372.657,Z 851.403,A -85,B 0,C 180,E1 -20782.968,E2 -20782.968} C_VEL
LIN {X 0,Y 373.886,Z 852.06,A -85,B 0,C 180,E1 -20785.688,E2 -20785.688} C_VEL
LIN {X 0,Y 374.478,Z 852.22,A -85,B 0,C 180,E1 -20787.849,E2 -20787.849} C_VEL
LIN {X 0,Y 374.688,Z 852.374,A -85,B 0,C 180,E1 -20790,E2 -20790} C_VEL
LIN {X 0,Y 374.478,Z 852.219,A -85,B 0,C 180,E1 -20792.151,E2 -20792.151} C_VEL
LIN {X 0,Y 373.757,Z 851.939,A -85,B 0,C 180,E1 -20794.739,E2 -20794.739} C_VEL
LIN {X 0,Y 372.668,Z 851.308,A -85,B 0,C 180,E1 -20797.033,E2 -20797.033} C_VEL
LIN {X 0,Y 370.776,Z 850.508,A -85,B 0,C 180,E1 -20799.822,E2 -20799.822} C_VEL
LIN {X 0,Y 368.636,Z 849.178,A -85,B 0,C 180,E1 -20802.237,E2 -20802.237} C_VEL
LIN {X 0,Y 366.124,Z 847.104,A -85,B 0,C 180,E1 -20804.693,E2 -20804.693} C_VEL
LIN {X 0,Y 363.085,Z 844.08,A -85,B 0,C 180,E1 -20807.233,E2 -20807.233} C_VEL
LIN {X 0,Y 359.635,Z 842.016,A -85,B 0,C 180,E1 -20809.63,E2 -20809.63} C_VEL
LIN {X 0,Y 355.723,Z 838.831,A -85,B 0,C 180,E1 -20812.136,E2 -20812.136} C_VEL
LIN {X 0,Y 352.948,Z 836.236,A -85,B 0,C 180,E1 -20813.781,E2 -20813.781} C_VEL
LIN {X 0,Y 348.252,Z 832.962,A -85,B 0,C 180,E1 -20816.297,E2 -20816.297} C_VEL
LIN {X 0,Y 343.101,Z 828.283,A -85,B 0,C 180,E1 -20818.895,E2 -20818.895} C_VEL
LIN {X 0,Y 338.313,Z 824.475,A -85,B 0,C 180,E1 -20821.123,E2 -20821.123} C_VEL
LIN {X 0,Y 333.936,Z 820.547,A -85,B 0,C 180,E1 -20823.069,E2 -20823.069} C_VEL
LIN {X 0,Y 328.55,Z 815.888,A -85,B 0,C 180,E1 -20825.35,E2 -20825.35} C_VEL
LIN {X 0,Y 324.883,Z 812.741,A -85,B 0,C 180,E1 -20826.833,E2 -20826.833} C_VEL
LIN {X 0,Y 319.423,Z 807.805,A -85,B 0,C 180,E1 -20828.993,E2 -20828.993} C_VEL
LIN {X 0,Y 313.039,Z 802.149,A -85,B 0,C 180,E1 -20831.379,E2 -20831.379} C_VEL
LIN {X 0,Y 308.533,Z 798.12,A -85,B 0,C 180,E1 -20832.978,E2 -20832.978} C_VEL
LIN {X 0,Y 301.456,Z 791.845,A -85,B 0,C 180,E1 -20835.261,E2 -20835.261} C_VEL
LIN {X 0,Y 293.789,Z 785.224,A -85,B 0,C 180,E1 -20837.513,E2 -20837.513} C_VEL
LIN {X 0,Y 287.92,Z 780.049,A -85,B 0,C 180,E1 -20839.131,E2 -20839.131} C_VEL
LIN {X 0,Y 280.067,Z 772.975,A -85,B 0,C 180,E1 -20841.323,E2 -20841.323} C_VEL
LIN {X 0,Y 272.168,Z 764.37,A -85,B 0,C 180,E1 -20843.844,E2 -20843.844} C_VEL
LIN {X 0,Y 266.57,Z 757.282,A -85,B 0,C 180,E1 -20845.871,E2 -20845.871} C_VEL
LIN {X 0,Y 256.903,Z 743.22,A -85,B 0,C 180,E1 -20849.99,E2 -20849.99} C_VEL
LIN {X 0,Y 253.183,Z 738.169,A -85,B 0,C 180,E1 -20851.791,E2 -20851.791} C_VEL
LIN {X 0,Y 250.305,Z 734.204,A -85,B 0,C 180,E1 -20853.305,E2 -20853.305} C_VEL
LIN {X 0,Y 247.331,Z 730.146,A -85,B 0,C 180,E1 -20854.997,E2 -20854.997} C_VEL
LIN {X 0,Y 244.264,Z 726.019,A -85,B 0,C 180,E1 -20856.906,E2 -20856.906} C_VEL
LIN {X 0,Y 241.13,Z 722.521,A -85,B 0,C 180,E1 -20859.026,E2 -20859.026} C_VEL
LIN {X 0,Y 240.032,Z 720.778,A -85,B 0,C 180,E1 -20859.878,E2 -20859.878} C_VEL
LIN {X 0,Y 237.24,Z 717.981,A -85,B 0,C 180,E1 -20862.101,E2 -20862.101} C_VEL
LIN {X 0,Y 235.683,Z 715.36,A -85,B 0,C 180,E1 -20863.608,E2 -20863.608} C_VEL
LIN {X 0,Y 232.977,Z 713.146,A -85,B 0,C 180,E1 -20866.369,E2 -20866.369} C_VEL
LIN {X 0,Y 231.222,Z 709.978,A -85,B 0,C 180,E1 -20868.828,E2 -20868.828} C_VEL
LIN {X 0,Y 227.485,Z 706.146,A -85,B 0,C 180,E1 -20879.115,E2 -20879.115} C_VEL
LIN {X 0,Y 227.532,Z 706.296,A -85,B 0,C 180,E1 -20881.328,E2 -20881.328} C_VEL
LIN {X 0,Y 231.427,Z 710.159,A -85,B 0,C 180,E1 -20891.052,E2 -20891.052} C_VEL
LIN {X 0,Y 233.039,Z 713.21,A -85,B 0,C 180,E1 -20893.295,E2 -20893.295} C_VEL
LIN {X 0,Y 236.005,Z 715.82,A -85,B 0,C 180,E1 -20896.301,E2 -20896.301} C_VEL
LIN {X 0,Y 238.146,Z 719.171,A -85,B 0,C 180,E1 -20898.274,E2 -20898.274} C_VEL
LIN {X 0,Y 240.437,Z 721.391,A -85,B 0,C 180,E1 -20900.032,E2 -20900.032} C_VEL
LIN {X 0,Y 242.966,Z 724.839,A -85,B 0,C 180,E1 -20901.86,E2 -20901.86} C_VEL
LIN {X 0,Y 244.478,Z 726.431,A -85,B 0,C 180,E1 -20902.836,E2 -20902.836} C_VEL
LIN {X 0,Y 248.479,Z 731.726,A -85,B 0,C 180,E1 -20905.267,E2 -20905.267} C_VEL
LIN {X 0,Y 252.147,Z 736.727,A -85,B 0,C 180,E1 -20907.268,E2 -20907.268} C_VEL
LIN {X 0,Y 255.779,Z 741.748,A -85,B 0,C 180,E1 -20909.078,E2 -20909.078} C_VEL
LIN {X 0,Y 260.832,Z 750.556,A -85,B 0,C 180,E1 -20911.456,E2 -20911.456} C_VEL
LIN {X 0,Y 266.426,Z 761.13,A -85,B 0,C 180,E1 -20913.858,E2 -20913.858} C_VEL
LIN {X 0,Y 271.76,Z 772.349,A -85,B 0,C 180,E1 -20915.982,E2 -20915.982} C_VEL
LIN {X 0,Y 276.588,Z 783.349,A -85,B 0,C 180,E1 -20917.785,E2 -20917.785} C_VEL
LIN {X 0,Y 277.119,Z 785.067,A -85,B 0,C 180,E1 -20917.996,E2 -20917.996} C_VEL
LIN {X 0,Y 270.134,Z 889.048,A -85,B 0,C 180,E1 -20920.489,E2 -20920.489} C_VEL
LIN {X 0,Y 268.736,Z 901.706,A -85,B 0,C 180,E1 -20920.921,E2 -20920.921} C_VEL
LIN {X 0,Y 267.028,Z 912.737,A -85,B 0,C 180,E1 -20921.385,E2 -20921.385} C_VEL
LIN {X 0,Y 265.737,Z 916.537,A -85,B 0,C 180,E1 -20921.429,E2 -20921.429} C_VEL
LIN {X 0,Y 259.864,Z 927.341,A -85,B 0,C 180,E1 -20921.155,E2 -20921.155} C_VEL
LIN {X 0,Y 258.476,Z 930.863,A -85,B 0,C 180,E1 -20921.252,E2 -20921.252} C_VEL
LIN {X 0,Y 258.168,Z 932.104,A -85,B 0,C 180,E1 -20921.329,E2 -20921.329} C_VEL
LIN {X 0,Y 254.107,Z 947.813,A -85,B 0,C 180,E1 -20922.577,E2 -20922.577} C_VEL
LIN {X 0,Y 249.409,Z 962.476,A -85,B 0,C 180,E1 -20924.066,E2 -20924.066} C_VEL
LIN {X 0,Y 244.939,Z 974.905,A -85,B 0,C 180,E1 -20925.624,E2 -20925.624} C_VEL
LIN {X 0,Y 240.559,Z 986.146,A -85,B 0,C 180,E1 -20927.332,E2 -20927.332} C_VEL
LIN {X 0,Y 236.103,Z 996.19,A -85,B 0,C 180,E1 -20929.092,E2 -20929.092} C_VEL
LIN {X 0,Y 231.921,Z 1005.458,A -85,B 0,C 180,E1 -20931.04,E2 -20931.04} C_VEL
LIN {X 0,Y 226.737,Z 1016.058,A -85,B 0,C 180,E1 -20933.698,E2 -20933.698} C_VEL
LIN {X 0,Y 222.267,Z 1024.989,A -85,B 0,C 180,E1 -20936.404,E2 -20936.404} C_VEL
LIN {X 0,Y 218.467,Z 1032.308,A -85,B 0,C 180,E1 -20939.023,E2 -20939.023} C_VEL
LIN {X 0,Y 214.749,Z 1039.478,A -85,B 0,C 180,E1 -20942.082,E2 -20942.082} C_VEL
LIN {X 0,Y 211.481,Z 1046.007,A -85,B 0,C 180,E1 -20945.456,E2 -20945.456} C_VEL
LIN {X 0,Y 209.218,Z 1050.662,A -85,B 0,C 180,E1 -20948.315,E2 -20948.315} C_VEL
LIN {X 0,Y 206.945,Z 1055.769,A -85,B 0,C 180,E1 -20952.203,E2 -20952.203} C_VEL
LIN {X 0,Y 205.409,Z 1059.779,A -85,B 0,C 180,E1 -20956.143,E2 -20956.143} C_VEL
LIN {X 0,Y 204.577,Z 1062.749,A -85,B 0,C 180,E1 -20960.11,E2 -20960.11} C_VEL
LIN {X 0,Y 204.382,Z 1063.942,A -85,B 0,C 180,E1 -20962.094,E2 -20962.094} C_VEL
LIN {X 0,Y 204.261,Z 1065.461,A -85,B 0,C 180,E1 -20966.201,E2 -20966.201} C_VEL
LIN {X 0,Y 204.463,Z 1065.921,A -85,B 0,C 180,E1 -20970,E2 -20970} C_VEL
LIN {X 0,Y 204.264,Z 1065.423,A -85,B 0,C 180,E1 -20973.946,E2 -20973.946} C_VEL
LIN {X 0,Y 204.382,Z 1063.942,A -85,B 0,C 180,E1 -20977.906,E2 -20977.906} C_VEL
LIN {X 0,Y 204.891,Z 1061.459,A -85,B 0,C 180,E1 -20981.876,E2 -20981.876} C_VEL
LIN {X 0,Y 206.534,Z 1056.861,A -85,B 0,C 180,E1 -20986.812,E2 -20986.812} C_VEL
LIN {X 0,Y 208.576,Z 1052.013,A -85,B 0,C 180,E1 -20990.719,E2 -20990.719} C_VEL
LIN {X 0,Y 210.662,Z 1047.63,A -85,B 0,C 180,E1 -20993.599,E2 -20993.599} C_VEL
LIN {X 0,Y 213.223,Z 1042.566,A -85,B 0,C 180,E1 -20996.421,E2 -20996.421} C_VEL
LIN {X 0,Y 217.322,Z 1034.531,A -85,B 0,C 180,E1 -21000.082,E2 -21000.082} C_VEL
LIN {X 0,Y 220.945,Z 1027.547,A -85,B 0,C 180,E1 -21002.734,E2 -21002.734} C_VEL
LIN {X 0,Y 225.039,Z 1019.582,A -85,B 0,C 180,E1 -21005.292,E2 -21005.292} C_VEL
LIN {X 0,Y 229.499,Z 1010.471,A -85,B 0,C 180,E1 -21007.767,E2 -21007.767} C_VEL
LIN {X 0,Y 233.532,Z 1001.906,A -85,B 0,C 180,E1 -21009.754,E2 -21009.754} C_VEL
LIN {X 0,Y 238.345,Z 991.135,A -85,B 0,C 180,E1 -21011.845,E2 -21011.845} C_VEL
LIN {X 0,Y 243.141,Z 979.493,A -85,B 0,C 180,E1 -21013.728,E2 -21013.728} C_VEL
LIN {X 0,Y 247.398,Z 968.226,A -85,B 0,C 180,E1 -21015.249,E2 -21015.249} C_VEL
LIN {X 0,Y 251.477,Z 956.208,A -85,B 0,C 180,E1 -21016.602,E2 -21016.602} C_VEL
LIN {X 0,Y 255.146,Z 943.894,A -85,B 0,C 180,E1 -21017.753,E2 -21017.753} C_VEL
LIN {X 0,Y 258.355,Z 931.354,A -85,B 0,C 180,E1 -21018.717,E2 -21018.717} C_VEL
LIN {X 0,Y 261.242,Z 918.257,A -85,B 0,C 180,E1 -21019.503,E2 -21019.503} C_VEL
LIN {X 0,Y 263.614,Z 904.875,A -85,B 0,C 180,E1 -21020.123,E2 -21020.123} C_VEL
LIN {X 0,Y 265.316,Z 891.888,A -85,B 0,C 180,E1 -21020.577,E2 -21020.577} C_VEL
LIN {X 0,Y 267.291,Z 865.164,A -85,B 0,C 180,E1 -21021.278,E2 -21021.278} C_VEL
LIN {X 0,Y 272.615,Z 787.299,A -85,B 0,C 180,E1 -21023.128,E2 -21023.128} C_VEL
LIN {X 0,Y 266.911,Z 774.128,A -85,B 0,C 180,E1 -21025.384,E2 -21025.384} C_VEL
LIN {X 0,Y 261.751,Z 763.325,A -85,B 0,C 180,E1 -21027.577,E2 -21027.577} C_VEL
LIN {X 0,Y 255.947,Z 752.352,A -85,B 0,C 180,E1 -21030.266,E2 -21030.266} C_VEL
LIN {X 0,Y 252.462,Z 746.377,A -85,B 0,C 180,E1 -21032.02,E2 -21032.02} C_VEL
LIN {X 0,Y 248.184,Z 740.475,A -85,B 0,C 180,E1 -21034.303,E2 -21034.303} C_VEL
LIN {X 0,Y 244.967,Z 736.091,A -85,B 0,C 180,E1 -21036.206,E2 -21036.206} C_VEL
LIN {X 0,Y 241.977,Z 732.12,A -85,B 0,C 180,E1 -21038.154,E2 -21038.154} C_VEL
LIN {X 0,Y 239.085,Z 728.53,A -85,B 0,C 180,E1 -21040.242,E2 -21040.242} C_VEL
LIN {X 0,Y 238.296,Z 727.371,A -85,B 0,C 180,E1 -21040.874,E2 -21040.874} C_VEL
LIN {X 0,Y 235.584,Z 724.373,A -85,B 0,C 180,E1 -21043.154,E2 -21043.154} C_VEL
LIN {X 0,Y 234.41,Z 722.275,A -85,B 0,C 180,E1 -21044.345,E2 -21044.345} C_VEL
LIN {X 0,Y 231.647,Z 719.809,A -85,B 0,C 180,E1 -21047.293,E2 -21047.293} C_VEL
LIN {X 0,Y 230.199,Z 716.869,A -85,B 0,C 180,E1 -21049.445,E2 -21049.445} C_VEL
LIN {X 0,Y 226.62,Z 713.072,A -85,B 0,C 180,E1 -21060,E2 -21060} C_VEL
LIN {X 0,Y 226.762,Z 713.929,A -85,B 0,C 180,E1 -21062.886,E2 -21062.886} C_VEL
LIN {X 0,Y 230.283,Z 717.081,A -85,B 0,C 180,E1 -21071.107,E2 -21071.107} C_VEL
LIN {X 0,Y 231.891,Z 720.131,A -85,B 0,C 180,E1 -21073.417,E2 -21073.417} C_VEL
LIN {X 0,Y 234.668,Z 722.687,A -85,B 0,C 180,E1 -21076.327,E2 -21076.327} C_VEL
LIN {X 0,Y 237.151,Z 726.344,A -85,B 0,C 180,E1 -21078.632,E2 -21078.632} C_VEL
LIN {X 0,Y 238.759,Z 727.94,A -85,B 0,C 180,E1 -21079.897,E2 -21079.897} C_VEL
LIN {X 0,Y 241.739,Z 731.87,A -85,B 0,C 180,E1 -21082.094,E2 -21082.094} C_VEL
LIN {X 0,Y 242.982,Z 733.404,A -85,B 0,C 180,E1 -21082.927,E2 -21082.927} C_VEL
LIN {X 0,Y 246.513,Z 738.186,A -85,B 0,C 180,E1 -21085.139,E2 -21085.139} C_VEL
LIN {X 0,Y 250.296,Z 743.486,A -85,B 0,C 180,E1 -21087.27,E2 -21087.27} C_VEL
LIN {X 0,Y 255.077,Z 750.109,A -85,B 0,C 180,E1 -21089.675,E2 -21089.675} C_VEL
LIN {X 0,Y 267.903,Z 768.645,A -85,B 0,C 180,E1 -21095.076,E2 -21095.076} C_VEL
LIN {X 0,Y 275.607,Z 777.284,A -85,B 0,C 180,E1 -21097.676,E2 -21097.676} C_VEL
LIN {X 0,Y 283.029,Z 784.482,A -85,B 0,C 180,E1 -21099.876,E2 -21099.876} C_VEL
LIN {X 0,Y 291.697,Z 791.918,A -85,B 0,C 180,E1 -21102.23,E2 -21102.23} C_VEL
LIN {X 0,Y 299.601,Z 798.644,A -85,B 0,C 180,E1 -21104.507,E2 -21104.507} C_VEL
LIN {X 0,Y 306.874,Z 805.022,A -85,B 0,C 180,E1 -21106.834,E2 -21106.834} C_VEL
LIN {X 0,Y 311.414,Z 809.039,A -85,B 0,C 180,E1 -21108.4,E2 -21108.4} C_VEL
LIN {X 0,Y 318.795,Z 815.604,A -85,B 0,C 180,E1 -21111.164,E2 -21111.164} C_VEL
LIN {X 0,Y 324.261,Z 820.307,A -85,B 0,C 180,E1 -21113.314,E2 -21113.314} C_VEL
LIN {X 0,Y 330.94,Z 826.182,A -85,B 0,C 180,E1 -21116.07,E2 -21116.07} C_VEL
LIN {X 0,Y 334.636,Z 829.237,A -85,B 0,C 180,E1 -21117.658,E2 -21117.658} C_VEL
LIN {X 0,Y 339.742,Z 833.74,A -85,B 0,C 180,E1 -21119.98,E2 -21119.98} C_VEL
LIN {X 0,Y 343.328,Z 836.494,A -85,B 0,C 180,E1 -21121.667,E2 -21121.667} C_VEL
LIN {X 0,Y 347.565,Z 840.279,A -85,B 0,C 180,E1 -21123.827,E2 -21123.827} C_VEL
LIN {X 0,Y 352.023,Z 843.369,A -85,B 0,C 180,E1 -21126.217,E2 -21126.217} C_VEL
LIN {X 0,Y 355.852,Z 846.882,A -85,B 0,C 180,E1 -21128.508,E2 -21128.508} C_VEL
LIN {X 0,Y 359.777,Z 849.827,A -85,B 0,C 180,E1 -21131.051,E2 -21131.051} C_VEL
LIN {X 0,Y 362.61,Z 851.515,A -85,B 0,C 180,E1 -21133.099,E2 -21133.099} C_VEL
LIN {X 0,Y 365.371,Z 854.34,A -85,B 0,C 180,E1 -21135.429,E2 -21135.429} C_VEL
LIN {X 0,Y 367.86,Z 856.296,A -85,B 0,C 180,E1 -21137.869,E2 -21137.869} C_VEL
LIN {X 0,Y 369.887,Z 857.548,A -85,B 0,C 180,E1 -21140.154,E2 -21140.154} C_VEL
LIN {X 0,Y 371.438,Z 858.255,A -85,B 0,C 180,E1 -21142.389,E2 -21142.389} C_VEL
LIN {X 0,Y 372.602,Z 858.79,A -85,B 0,C 180,E1 -21144.589,E2 -21144.589} C_VEL
LIN {X 0,Y 373.385,Z 859.22,A -85,B 0,C 180,E1 -21146.763,E2 -21146.763} C_VEL
LIN {X 0,Y 373.74,Z 859.352,A -85,B 0,C 180,E1 -21148.923,E2 -21148.923} C_VEL
LIN {X 0,Y 373.74,Z 859.352,A -85,B 0,C 180,E1 -21151.077,E2 -21151.077} C_VEL
LIN {X 0,Y 373.248,Z 859.157,A -85,B 0,C 180,E1 -21153.678,E2 -21153.678} C_VEL
LIN {X 0,Y 372.31,Z 858.625,A -85,B 0,C 180,E1 -21156.034,E2 -21156.034} C_VEL
LIN {X 0,Y 370.719,Z 857.811,A -85,B 0,C 180,E1 -21158.723,E2 -21158.723} C_VEL
LIN {X 0,Y 368.917,Z 857.023,A -85,B 0,C 180,E1 -21160.982,E2 -21160.982} C_VEL
LIN {X 0,Y 366.355,Z 855.189,A -85,B 0,C 180,E1 -21163.637,E2 -21163.637} C_VEL
LIN {X 0,Y 363.53,Z 852.529,A -85,B 0,C 180,E1 -21166.168,E2 -21166.168} C_VEL
LIN {X 0,Y 361.713,Z 850.893,A -85,B 0,C 180,E1 -21167.596,E2 -21167.596} C_VEL
LIN {X 0,Y 358.144,Z 848.681,A -85,B 0,C 180,E1 -21170.026,E2 -21170.026} C_VEL
LIN {X 0,Y 354.177,Z 845.436,A -85,B 0,C 180,E1 -21172.51,E2 -21172.51} C_VEL
LIN {X 0,Y 351.68,Z 843.119,A -85,B 0,C 180,E1 -21173.974,E2 -21173.974} C_VEL
LIN {X 0,Y 346.857,Z 839.777,A -85,B 0,C 180,E1 -21176.531,E2 -21176.531} C_VEL
LIN {X 0,Y 341.661,Z 835.101,A -85,B 0,C 180,E1 -21179.126,E2 -21179.126} C_VEL
LIN {X 0,Y 336.811,Z 831.274,A -85,B 0,C 180,E1 -21181.358,E2 -21181.358} C_VEL
LIN {X 0,Y 332.074,Z 827.069,A -85,B 0,C 180,E1 -21183.455,E2 -21183.455} C_VEL
LIN {X 0,Y 326.54,Z 822.292,A -85,B 0,C 180,E1 -21185.765,E2 -21185.765} C_VEL
LIN {X 0,Y 319.68,Z 816.455,A -85,B 0,C 180,E1 -21188.486,E2 -21188.486} C_VEL
LIN {X 0,Y 314.175,Z 811.505,A -85,B 0,C 180,E1 -21190.589,E2 -21190.589} C_VEL
LIN {X 0,Y 307.643,Z 805.601,A -85,B 0,C 180,E1 -21192.914,E2 -21192.914} C_VEL
LIN {X 0,Y 302.032,Z 800.754,A -85,B 0,C 180,E1 -21194.722,E2 -21194.722} C_VEL
LIN {X 0,Y 294.488,Z 794.311,A -85,B 0,C 180,E1 -21196.992,E2 -21196.992} C_VEL
LIN {X 0,Y 286.135,Z 787.224,A -85,B 0,C 180,E1 -21199.276,E2 -21199.276} C_VEL
LIN {X 0,Y 276.898,Z 778.644,A -85,B 0,C 180,E1 -21201.92,E2 -21201.92} C_VEL
LIN {X 0,Y 269.541,Z 770.547,A -85,B 0,C 180,E1 -21204.342,E2 -21204.342} C_VEL
LIN {X 0,Y 261.52,Z 760.061,A -85,B 0,C 180,E1 -21207.413,E2 -21207.413} C_VEL
LIN {X 0,Y 254.513,Z 749.337,A -85,B 0,C 180,E1 -21210.594,E2 -21210.594} C_VEL
LIN {X 0,Y 248.504,Z 740.857,A -85,B 0,C 180,E1 -21213.719,E2 -21213.719} C_VEL
LIN {X 0,Y 245.196,Z 736.358,A -85,B 0,C 180,E1 -21215.66,E2 -21215.66} C_VEL
LIN {X 0,Y 241.887,Z 732.01,A -85,B 0,C 180,E1 -21217.809,E2 -21217.809} C_VEL
LIN {X 0,Y 238.946,Z 728.25,A -85,B 0,C 180,E1 -21219.951,E2 -21219.951} C_VEL
LIN {X 0,Y 237.983,Z 727.084,A -85,B 0,C 180,E1 -21220.709,E2 -21220.709} C_VEL
LIN {X 0,Y 235.277,Z 723.85,A -85,B 0,C 180,E1 -21223.047,E2 -21223.047} C_VEL
LIN {X 0,Y 234.279,Z 722.188,A -85,B 0,C 180,E1 -21224.061,E2 -21224.061} C_VEL
LIN {X 0,Y 231.677,Z 719.841,A -85,B 0,C 180,E1 -21226.85,E2 -21226.85} C_VEL
LIN {X 0,Y 230.067,Z 716.836,A -85,B 0,C 180,E1 -21229.217,E2 -21229.217} C_VEL
LIN {X 0,Y 226.618,Z 713.202,A -85,B 0,C 180,E1 -21239.112,E2 -21239.112} C_VEL
LIN {X 0,Y 226.663,Z 713.369,A -85,B 0,C 180,E1 -21241.333,E2 -21241.333} C_VEL
LIN {X 0,Y 230.26,Z 717.047,A -85,B 0,C 180,E1 -21250.664,E2 -21250.664} C_VEL
LIN {X 0,Y 232.078,Z 720.389,A -85,B 0,C 180,E1 -21253.239,E2 -21253.239} C_VEL
LIN {X 0,Y 234.615,Z 722.596,A -85,B 0,C 180,E1 -21255.865,E2 -21255.865} C_VEL
LIN {X 0,Y 236.737,Z 725.934,A -85,B 0,C 180,E1 -21257.883,E2 -21257.883} C_VEL
LIN {X 0,Y 238.743,Z 727.944,A -85,B 0,C 180,E1 -21259.48,E2 -21259.48} C_VEL
LIN {X 0,Y 241.642,Z 731.81,A -85,B 0,C 180,E1 -21261.624,E2 -21261.624} C_VEL
LIN {X 0,Y 242.854,Z 733.239,A -85,B 0,C 180,E1 -21262.435,E2 -21262.435} C_VEL
LIN {X 0,Y 246.629,Z 738.348,A -85,B 0,C 180,E1 -21264.8,E2 -21264.8} C_VEL
LIN {X 0,Y 250.214,Z 743.366,A -85,B 0,C 180,E1 -21266.819,E2 -21266.819} C_VEL
LIN {X 0,Y 253.237,Z 747.6,A -85,B 0,C 180,E1 -21268.377,E2 -21268.377} C_VEL
LIN {X 0,Y 258.564,Z 757.166,A -85,B 0,C 180,E1 -21270.98,E2 -21270.98} C_VEL
LIN {X 0,Y 264.358,Z 768.59,A -85,B 0,C 180,E1 -21273.548,E2 -21273.548} C_VEL
LIN {X 0,Y 270.515,Z 782.273,A -85,B 0,C 180,E1 -21276.059,E2 -21276.059} C_VEL
LIN {X 0,Y 272.613,Z 787.364,A -85,B 0,C 180,E1 -21276.874,E2 -21276.874} C_VEL
LIN {X 0,Y 265.647,Z 888.17,A -85,B 0,C 180,E1 -21279.303,E2 -21279.303} C_VEL
LIN {X 0,Y 264.19,Z 901.236,A -85,B 0,C 180,E1 -21279.751,E2 -21279.751} C_VEL
LIN {X 0,Y 262.082,Z 914.023,A -85,B 0,C 180,E1 -21280.291,E2 -21280.291} C_VEL
LIN {X 0,Y 259.471,Z 926.571,A -85,B 0,C 180,E1 -21280.975,E2 -21280.975} C_VEL
LIN {X 0,Y 258.168,Z 932.104,A -85,B 0,C 180,E1 -21281.329,E2 -21281.329} C_VEL
LIN {X 0,Y 256.502,Z 937.613,A -85,B 0,C 180,E1 -21281.628,E2 -21281.628} C_VEL
LIN {X 0,Y 252.172,Z 946.482,A -85,B 0,C 180,E1 -21281.869,E2 -21281.869} C_VEL
LIN {X 0,Y 247.466,Z 955.119,A -85,B 0,C 180,E1 -21282.192,E2 -21282.192} C_VEL
LIN {X 0,Y 245.229,Z 960.259,A -85,B 0,C 180,E1 -21282.63,E2 -21282.63} C_VEL
LIN {X 0,Y 239.87,Z 974.697,A -85,B 0,C 180,E1 -21284.427,E2 -21284.427} C_VEL
LIN {X 0,Y 235.917,Z 984.597,A -85,B 0,C 180,E1 -21285.919,E2 -21285.919} C_VEL
LIN {X 0,Y 230.737,Z 995.983,A -85,B 0,C 180,E1 -21287.927,E2 -21287.927} C_VEL
LIN {X 0,Y 226.378,Z 1005.25,A -85,B 0,C 180,E1 -21289.896,E2 -21289.896} C_VEL
LIN {X 0,Y 221.468,Z 1014.978,A -85,B 0,C 180,E1 -21292.349,E2 -21292.349} C_VEL
LIN {X 0,Y 217.044,Z 1023.502,A -85,B 0,C 180,E1 -21294.919,E2 -21294.919} C_VEL
LIN {X 0,Y 212.344,Z 1032.1,A -85,B 0,C 180,E1 -21298.026,E2 -21298.026} C_VEL
LIN {X 0,Y 208.723,Z 1038.718,A -85,B 0,C 180,E1 -21300.884,E2 -21300.884} C_VEL
LIN {X 0,Y 204.954,Z 1045.799,A -85,B 0,C 180,E1 -21304.62,E2 -21304.62} C_VEL
LIN {X 0,Y 202.54,Z 1050.454,A -85,B 0,C 180,E1 -21307.562,E2 -21307.562} C_VEL
LIN {X 0,Y 200.104,Z 1055.561,A -85,B 0,C 180,E1 -21311.574,E2 -21311.574} C_VEL
LIN {X 0,Y 198.442,Z 1059.571,A -85,B 0,C 180,E1 -21315.646,E2 -21315.646} C_VEL
LIN {X 0,Y 197.539,Z 1062.542,A -85,B 0,C 180,E1 -21319.753,E2 -21319.753} C_VEL
LIN {X 0,Y 197.305,Z 1063.735,A -85,B 0,C 180,E1 -21321.809,E2 -21321.809} C_VEL
LIN {X 0,Y 197.163,Z 1065.31,A -85,B 0,C 180,E1 -21326.447,E2 -21326.447} C_VEL
LIN {X 0,Y 197.363,Z 1065.715,A -85,B 0,C 180,E1 -21330,E2 -21330} C_VEL
LIN {X 0,Y 197.173,Z 1065.218,A -85,B 0,C 180,E1 -21334.088,E2 -21334.088} C_VEL
LIN {X 0,Y 197.305,Z 1063.735,A -85,B 0,C 180,E1 -21338.191,E2 -21338.191} C_VEL
LIN {X 0,Y 197.869,Z 1061.251,A -85,B 0,C 180,E1 -21342.304,E2 -21342.304} C_VEL
LIN {X 0,Y 199.643,Z 1056.653,A -85,B 0,C 180,E1 -21347.411,E2 -21347.411} C_VEL
LIN {X 0,Y 201.208,Z 1053.155,A -85,B 0,C 180,E1 -21350.443,E2 -21350.443} C_VEL
LIN {X 0,Y 204.071,Z 1047.421,A -85,B 0,C 180,E1 -21354.41,E2 -21354.41} C_VEL
LIN {X 0,Y 206.782,Z 1042.357,A -85,B 0,C 180,E1 -21357.311,E2 -21357.311} C_VEL
LIN {X 0,Y 211.102,Z 1034.322,A -85,B 0,C 180,E1 -21361.065,E2 -21361.065} C_VEL
LIN {X 0,Y 214.925,Z 1027.339,A -85,B 0,C 180,E1 -21363.771,E2 -21363.771} C_VEL
LIN {X 0,Y 219.633,Z 1018.483,A -85,B 0,C 180,E1 -21366.643,E2 -21366.643} C_VEL
LIN {X 0,Y 223.87,Z 1010.264,A -85,B 0,C 180,E1 -21368.892,E2 -21368.892} C_VEL
LIN {X 0,Y 228.064,Z 1001.698,A -85,B 0,C 180,E1 -21370.906,E2 -21370.906} C_VEL
LIN {X 0,Y 233.071,Z 990.928,A -85,B 0,C 180,E1 -21373.017,E2 -21373.017} C_VEL
LIN {X 0,Y 237.63,Z 980.255,A -85,B 0,C 180,E1 -21374.78,E2 -21374.78} C_VEL
LIN {X 0,Y 242.408,Z 968.019,A -85,B 0,C 180,E1 -21376.452,E2 -21376.452} C_VEL
LIN {X 0,Y 246.628,Z 956.001,A -85,B 0,C 180,E1 -21377.807,E2 -21377.807} C_VEL
LIN {X 0,Y 250.411,Z 943.688,A -85,B 0,C 180,E1 -21378.96,E2 -21378.96} C_VEL
LIN {X 0,Y 253.705,Z 931.148,A -85,B 0,C 180,E1 -21379.928,E2 -21379.928} C_VEL
LIN {X 0,Y 256.765,Z 917.696,A -85,B 0,C 180,E1 -21380.725,E2 -21380.725} C_VEL
LIN {X 0,Y 259.081,Z 904.875,A -85,B 0,C 180,E1 -21381.322,E2 -21381.322} C_VEL
LIN {X 0,Y 260.864,Z 891.682,A -85,B 0,C 180,E1 -21381.782,E2 -21381.782} C_VEL
LIN {X 0,Y 262.9,Z 864.958,A -85,B 0,C 180,E1 -21382.488,E2 -21382.488} C_VEL
LIN {X 0,Y 268.179,Z 789.925,A -85,B 0,C 180,E1 -21384.284,E2 -21384.284} C_VEL
LIN {X 0,Y 262.231,Z 776.078,A -85,B 0,C 180,E1 -21386.788,E2 -21386.788} C_VEL
LIN {X 0,Y 257.313,Z 765.806,A -85,B 0,C 180,E1 -21389.024,E2 -21389.024} C_VEL
LIN {X 0,Y 252.385,Z 756.465,A -85,B 0,C 180,E1 -21391.462,E2 -21391.462} C_VEL
LIN {X 0,Y 249.603,Z 751.696,A -85,B 0,C 180,E1 -21392.941,E2 -21392.941} C_VEL
LIN {X 0,Y 243.514,Z 743.022,A -85,B 0,C 180,E1 -21396.483,E2 -21396.483} C_VEL
LIN {X 0,Y 239.963,Z 738.398,A -85,B 0,C 180,E1 -21398.862,E2 -21398.862} C_VEL
LIN {X 0,Y 237.077,Z 734.44,A -85,B 0,C 180,E1 -21401.08,E2 -21401.08} C_VEL
LIN {X 0,Y 233.801,Z 730.528,A -85,B 0,C 180,E1 -21403.966,E2 -21403.966} C_VEL
LIN {X 0,Y 232.905,Z 729.005,A -85,B 0,C 180,E1 -21404.915,E2 -21404.915} C_VEL
LIN {X 0,Y 230.123,Z 726.171,A -85,B 0,C 180,E1 -21408.103,E2 -21408.103} C_VEL
LIN {X 0,Y 228.933,Z 723.728,A -85,B 0,C 180,E1 -21409.997,E2 -21409.997} C_VEL
LIN {X 0,Y 225.754,Z 720.123,A -85,B 0,C 180,E1 -21420,E2 -21420} C_VEL
LIN {X 0,Y 225.89,Z 721.034,A -85,B 0,C 180,E1 -21422.897,E2 -21422.897} C_VEL
LIN {X 0,Y 229.126,Z 723.968,A -85,B 0,C 180,E1 -21430.716,E2 -21430.716} C_VEL
LIN {X 0,Y 230.804,Z 727.14,A -85,B 0,C 180,E1 -21433.201,E2 -21433.201} C_VEL
LIN {X 0,Y 233.274,Z 729.451,A -85,B 0,C 180,E1 -21435.871,E2 -21435.871} C_VEL
LIN {X 0,Y 235.865,Z 733.245,A -85,B 0,C 180,E1 -21438.344,E2 -21438.344} C_VEL
LIN {X 0,Y 237.306,Z 734.799,A -85,B 0,C 180,E1 -21439.517,E2 -21439.517} C_VEL
LIN {X 0,Y 240.266,Z 738.663,A -85,B 0,C 180,E1 -21441.75,E2 -21441.75} C_VEL
LIN {X 0,Y 244.405,Z 744.348,A -85,B 0,C 180,E1 -21444.488,E2 -21444.488} C_VEL
LIN {X 0,Y 248.197,Z 749.844,A -85,B 0,C 180,E1 -21446.712,E2 -21446.712} C_VEL
LIN {X 0,Y 252.792,Z 756.441,A -85,B 0,C 180,E1 -21449.112,E2 -21449.112} C_VEL
LIN {X 0,Y 265.399,Z 774.913,A -85,B 0,C 180,E1 -21454.588,E2 -21454.588} C_VEL
LIN {X 0,Y 273.004,Z 783.527,A -85,B 0,C 180,E1 -21457.226,E2 -21457.226} C_VEL
LIN {X 0,Y 280.165,Z 790.584,A -85,B 0,C 180,E1 -21459.407,E2 -21459.407} C_VEL
LIN {X 0,Y 289.586,Z 798.609,A -85,B 0,C 180,E1 -21461.974,E2 -21461.974} C_VEL
LIN {X 0,Y 296.726,Z 804.692,A -85,B 0,C 180,E1 -21464.008,E2 -21464.008} C_VEL
LIN {X 0,Y 304.08,Z 810.946,A -85,B 0,C 180,E1 -21466.267,E2 -21466.267} C_VEL
LIN {X 0,Y 309.893,Z 816.054,A -85,B 0,C 180,E1 -21468.231,E2 -21468.231} C_VEL
LIN {X 0,Y 316.749,Z 822.052,A -85,B 0,C 180,E1 -21470.769,E2 -21470.769} C_VEL
LIN {X 0,Y 322.36,Z 826.86,A -85,B 0,C 180,E1 -21472.956,E2 -21472.956} C_VEL
LIN {X 0,Y 329.245,Z 832.853,A -85,B 0,C 180,E1 -21475.768,E2 -21475.768} C_VEL
LIN {X 0,Y 333.201,Z 836.127,A -85,B 0,C 180,E1 -21477.461,E2 -21477.461} C_VEL
LIN {X 0,Y 338.362,Z 840.61,A -85,B 0,C 180,E1 -21479.787,E2 -21479.787} C_VEL
LIN {X 0,Y 341.812,Z 843.242,A -85,B 0,C 180,E1 -21481.397,E2 -21481.397} C_VEL
LIN {X 0,Y 346.168,Z 847.099,A -85,B 0,C 180,E1 -21483.592,E2 -21483.592} C_VEL
LIN {X 0,Y 350.836,Z 850.308,A -85,B 0,C 180,E1 -21486.068,E2 -21486.068} C_VEL
LIN {X 0,Y 354.706,Z 853.827,A -85,B 0,C 180,E1 -21488.353,E2 -21488.353} C_VEL
LIN {X 0,Y 358.804,Z 856.844,A -85,B 0,C 180,E1 -21490.998,E2 -21490.998} C_VEL
LIN {X 0,Y 361.65,Z 858.629,A -85,B 0,C 180,E1 -21493.053,E2 -21493.053} C_VEL
LIN {X 0,Y 364.548,Z 861.496,A -85,B 0,C 180,E1 -21495.486,E2 -21495.486} C_VEL
LIN {X 0,Y 366.95,Z 863.351,A -85,B 0,C 180,E1 -21497.838,E2 -21497.838} C_VEL
LIN {X 0,Y 368.997,Z 864.59,A -85,B 0,C 180,E1 -21500.13,E2 -21500.13} C_VEL
LIN {X 0,Y 370.556,Z 865.301,A -85,B 0,C 180,E1 -21502.371,E2 -21502.371} C_VEL
LIN {X 0,Y 371.727,Z 865.829,A -85,B 0,C 180,E1 -21504.576,E2 -21504.576} C_VEL
LIN {X 0,Y 372.521,Z 866.25,A -85,B 0,C 180,E1 -21506.756,E2 -21506.756} C_VEL
LIN {X 0,Y 372.873,Z 866.398,A -85,B 0,C 180,E1 -21508.92,E2 -21508.92} C_VEL
LIN {X 0,Y 372.873,Z 866.398,A -85,B 0,C 180,E1 -21511.08,E2 -21511.08} C_VEL
LIN {X 0,Y 372.521,Z 866.252,A -85,B 0,C 180,E1 -21513.244,E2 -21513.244} C_VEL
LIN {X 0,Y 371.727,Z 865.831,A -85,B 0,C 180,E1 -21515.424,E2 -21515.424} C_VEL
LIN {X 0,Y 370.558,Z 865.291,A -85,B 0,C 180,E1 -21517.629,E2 -21517.629} C_VEL
LIN {X 0,Y 368.73,Z 864.436,A -85,B 0,C 180,E1 -21520.172,E2 -21520.172} C_VEL
LIN {X 0,Y 366.425,Z 862.983,A -85,B 0,C 180,E1 -21522.732,E2 -21522.732} C_VEL
LIN {X 0,Y 363.723,Z 860.771,A -85,B 0,C 180,E1 -21525.219,E2 -21525.219} C_VEL
LIN {X 0,Y 361.005,Z 858.027,A -85,B 0,C 180,E1 -21527.463,E2 -21527.463} C_VEL
LIN {X 0,Y 357.366,Z 855.896,A -85,B 0,C 180,E1 -21529.941,E2 -21529.941} C_VEL
LIN {X 0,Y 353.389,Z 852.694,A -85,B 0,C 180,E1 -21532.433,E2 -21532.433} C_VEL
LIN {X 0,Y 350.348,Z 849.965,A -85,B 0,C 180,E1 -21534.208,E2 -21534.208} C_VEL
LIN {X 0,Y 345.509,Z 846.606,A -85,B 0,C 180,E1 -21536.746,E2 -21536.746} C_VEL
LIN {X 0,Y 340.005,Z 841.76,A -85,B 0,C 180,E1 -21539.466,E2 -21539.466} C_VEL
LIN {X 0,Y 335.109,Z 837.904,A -85,B 0,C 180,E1 -21541.688,E2 -21541.688} C_VEL
LIN {X 0,Y 330.517,Z 833.855,A -85,B 0,C 180,E1 -21543.696,E2 -21543.696} C_VEL
LIN {X 0,Y 324.792,Z 828.949,A -85,B 0,C 180,E1 -21546.071,E2 -21546.071} C_VEL
LIN {X 0,Y 317.7,Z 822.943,A -85,B 0,C 180,E1 -21548.864,E2 -21548.864} C_VEL
LIN {X 0,Y 312.067,Z 817.99,A -85,B 0,C 180,E1 -21550.961,E2 -21550.961} C_VEL
LIN {X 0,Y 306.965,Z 813.278,A -85,B 0,C 180,E1 -21552.778,E2 -21552.778} C_VEL
LIN {X 0,Y 301.325,Z 808.634,A -85,B 0,C 180,E1 -21554.586,E2 -21554.586} C_VEL
LIN {X 0,Y 296.199,Z 804.243,A -85,B 0,C 180,E1 -21556.147,E2 -21556.147} C_VEL
LIN {X 0,Y 288.327,Z 797.615,A -85,B 0,C 180,E1 -21558.365,E2 -21558.365} C_VEL
LIN {X 0,Y 274.707,Z 785.385,A -85,B 0,C 180,E1 -21562.228,E2 -21562.228} C_VEL
LIN {X 0,Y 266.264,Z 775.908,A -85,B 0,C 180,E1 -21565.095,E2 -21565.095} C_VEL
LIN {X 0,Y 258.525,Z 765.463,A -85,B 0,C 180,E1 -21568.194,E2 -21568.194} C_VEL
LIN {X 0,Y 252.066,Z 755.342,A -85,B 0,C 180,E1 -21571.253,E2 -21571.253} C_VEL
LIN {X 0,Y 245.968,Z 746.593,A -85,B 0,C 180,E1 -21574.566,E2 -21574.566} C_VEL
LIN {X 0,Y 242.919,Z 742.346,A -85,B 0,C 180,E1 -21576.446,E2 -21576.446} C_VEL
LIN {X 0,Y 240.261,Z 738.669,A -85,B 0,C 180,E1 -21578.252,E2 -21578.252} C_VEL
LIN {X 0,Y 237.245,Z 734.702,A -85,B 0,C 180,E1 -21580.534,E2 -21580.534} C_VEL
LIN {X 0,Y 233.698,Z 730.281,A -85,B 0,C 180,E1 -21583.673,E2 -21583.673} C_VEL
LIN {X 0,Y 232.945,Z 729.021,A -85,B 0,C 180,E1 -21584.47,E2 -21584.47} C_VEL
LIN {X 0,Y 230.31,Z 726.433,A -85,B 0,C 180,E1 -21587.443,E2 -21587.443} C_VEL
LIN {X 0,Y 229.063,Z 723.833,A -85,B 0,C 180,E1 -21589.393,E2 -21589.393} C_VEL
LIN {X 0,Y 225.754,Z 720.246,A -85,B 0,C 180,E1 -21599.109,E2 -21599.109} C_VEL
LIN {X 0,Y 225.796,Z 720.438,A -85,B 0,C 180,E1 -21601.338,E2 -21601.338} C_VEL
LIN {X 0,Y 229.119,Z 723.973,A -85,B 0,C 180,E1 -21610.3,E2 -21610.3} C_VEL
LIN {X 0,Y 230.902,Z 727.269,A -85,B 0,C 180,E1 -21612.916,E2 -21612.916} C_VEL
LIN {X 0,Y 233.307,Z 729.579,A -85,B 0,C 180,E1 -21615.507,E2 -21615.507} C_VEL
LIN {X 0,Y 235.878,Z 733.283,A -85,B 0,C 180,E1 -21617.951,E2 -21617.951} C_VEL
LIN {X 0,Y 237.257,Z 734.759,A -85,B 0,C 180,E1 -21619.073,E2 -21619.073} C_VEL
LIN {X 0,Y 240.252,Z 738.684,A -85,B 0,C 180,E1 -21621.336,E2 -21621.336} C_VEL
LIN {X 0,Y 244.613,Z 744.658,A -85,B 0,C 180,E1 -21624.211,E2 -21624.211} C_VEL
LIN {X 0,Y 250.124,Z 752.481,A -85,B 0,C 180,E1 -21627.338,E2 -21627.338} C_VEL
LIN {X 0,Y 254.356,Z 760.09,A -85,B 0,C 180,E1 -21629.54,E2 -21629.54} C_VEL
LIN {X 0,Y 259.887,Z 771.056,A -85,B 0,C 180,E1 -21632.168,E2 -21632.168} C_VEL
LIN {X 0,Y 264.905,Z 782.18,A -85,B 0,C 180,E1 -21634.366,E2 -21634.366} C_VEL
LIN {X 0,Y 268.194,Z 789.989,A -85,B 0,C 180,E1 -21635.724,E2 -21635.724} C_VEL
LIN {X 0,Y 261.078,Z 889.301,A -85,B 0,C 180,E1 -21638.139,E2 -21638.139} C_VEL
LIN {X 0,Y 259.564,Z 901.893,A -85,B 0,C 180,E1 -21638.575,E2 -21638.575} C_VEL
LIN {X 0,Y 257.468,Z 914.245,A -85,B 0,C 180,E1 -21639.109,E2 -21639.109} C_VEL
LIN {X 0,Y 254.862,Z 926.365,A -85,B 0,C 180,E1 -21639.767,E2 -21639.767} C_VEL
LIN {X 0,Y 252.062,Z 937.747,A -85,B 0,C 180,E1 -21640.557,E2 -21640.557} C_VEL
LIN {X 0,Y 248.238,Z 950.977,A -85,B 0,C 180,E1 -21641.695,E2 -21641.695} C_VEL
LIN {X 0,Y 245.229,Z 960.259,A -85,B 0,C 180,E1 -21642.63,E2 -21642.63} C_VEL
LIN {X 0,Y 242.941,Z 965.33,A -85,B 0,C 180,E1 -21643.107,E2 -21643.107} C_VEL
LIN {X 0,Y 233.528,Z 979.872,A -85,B 0,C 180,E1 -21644.153,E2 -21644.153} C_VEL
LIN {X 0,Y 230.801,Z 984.584,A -85,B 0,C 180,E1 -21644.725,E2 -21644.725} C_VEL
LIN {X 0,Y 230.078,Z 986.07,A -85,B 0,C 180,E1 -21644.974,E2 -21644.974} C_VEL
LIN {X 0,Y 225.467,Z 995.775,A -85,B 0,C 180,E1 -21646.706,E2 -21646.706} C_VEL
LIN {X 0,Y 220.91,Z 1005.041,A -85,B 0,C 180,E1 -21648.691,E2 -21648.691} C_VEL
LIN {X 0,Y 215.81,Z 1014.77,A -85,B 0,C 180,E1 -21651.18,E2 -21651.18} C_VEL
LIN {X 0,Y 211.175,Z 1023.293,A -85,B 0,C 180,E1 -21653.792,E2 -21653.792} C_VEL
LIN {X 0,Y 206.256,Z 1031.891,A -85,B 0,C 180,E1 -21656.964,E2 -21656.964} C_VEL
LIN {X 0,Y 202.442,Z 1038.514,A -85,B 0,C 180,E1 -21659.892,E2 -21659.892} C_VEL
LIN {X 0,Y 198.444,Z 1045.589,A -85,B 0,C 180,E1 -21663.725,E2 -21663.725} C_VEL
LIN {X 0,Y 195.89,Z 1050.245,A -85,B 0,C 180,E1 -21666.757,E2 -21666.757} C_VEL
LIN {X 0,Y 193.234,Z 1055.479,A -85,B 0,C 180,E1 -21671.021,E2 -21671.021} C_VEL
LIN {X 0,Y 191.499,Z 1059.364,A -85,B 0,C 180,E1 -21675.114,E2 -21675.114} C_VEL
LIN {X 0,Y 190.478,Z 1062.334,A -85,B 0,C 180,E1 -21679.369,E2 -21679.369} C_VEL
LIN {X 0,Y 190.226,Z 1063.528,A -85,B 0,C 180,E1 -21681.502,E2 -21681.502} C_VEL
LIN {X 0,Y 190.071,Z 1065.149,A -85,B 0,C 180,E1 -21686.701,E2 -21686.701} C_VEL
LIN {X 0,Y 190.266,Z 1065.51,A -85,B 0,C 180,E1 -21690,E2 -21690} C_VEL
LIN {X 0,Y 190.083,Z 1065.012,A -85,B 0,C 180,E1 -21694.241,E2 -21694.241} C_VEL
LIN {X 0,Y 190.226,Z 1063.528,A -85,B 0,C 180,E1 -21698.498,E2 -21698.498} C_VEL
LIN {X 0,Y 190.859,Z 1061.044,A -85,B 0,C 180,E1 -21702.764,E2 -21702.764} C_VEL
LIN {X 0,Y 192.758,Z 1056.507,A -85,B 0,C 180,E1 -21707.99,E2 -21707.99} C_VEL
LIN {X 0,Y 194.474,Z 1052.947,A -85,B 0,C 180,E1 -21711.185,E2 -21711.185} C_VEL
LIN {X 0,Y 197.531,Z 1047.212,A -85,B 0,C 180,E1 -21715.273,E2 -21715.273} C_VEL
LIN {X 0,Y 200.392,Z 1042.148,A -85,B 0,C 180,E1 -21718.258,E2 -21718.258} C_VEL
LIN {X 0,Y 204.348,Z 1035.225,A -85,B 0,C 180,E1 -21721.632,E2 -21721.632} C_VEL
LIN {X 0,Y 208.978,Z 1027.131,A -85,B 0,C 180,E1 -21724.869,E2 -21724.869} C_VEL
LIN {X 0,Y 213.17,Z 1019.667,A -85,B 0,C 180,E1 -21727.379,E2 -21727.379} C_VEL
LIN {X 0,Y 218.324,Z 1010.056,A -85,B 0,C 180,E1 -21730.075,E2 -21730.075} C_VEL
LIN {X 0,Y 222.672,Z 1001.49,A -85,B 0,C 180,E1 -21732.119,E2 -21732.119} C_VEL
LIN {X 0,Y 227.893,Z 990.721,A -85,B 0,C 180,E1 -21734.244,E2 -21734.244} C_VEL
LIN {X 0,Y 232.837,Z 979.566,A -85,B 0,C 180,E1 -21736.084,E2 -21736.084} C_VEL
LIN {X 0,Y 237.537,Z 967.812,A -85,B 0,C 180,E1 -21737.702,E2 -21737.702} C_VEL
LIN {X 0,Y 241.89,Z 955.795,A -85,B 0,C 180,E1 -21739.06,E2 -21739.06} C_VEL
LIN {X 0,Y 245.781,Z 943.481,A -85,B 0,C 180,E1 -21740.216,E2 -21740.216} C_VEL
LIN {X 0,Y 249.17,Z 930.942,A -85,B 0,C 180,E1 -21741.184,E2 -21741.184} C_VEL
LIN {X 0,Y 252.313,Z 917.543,A -85,B 0,C 180,E1 -21741.972,E2 -21741.972} C_VEL
LIN {X 0,Y 254.737,Z 904.381,A -85,B 0,C 180,E1 -21742.583,E2 -21742.583} C_VEL
LIN {X 0,Y 256.524,Z 891.477,A -85,B 0,C 180,E1 -21743.031,E2 -21743.031} C_VEL
LIN {X 0,Y 258.649,Z 864.753,A -85,B 0,C 180,E1 -21743.732,E2 -21743.732} C_VEL
LIN {X 0,Y 263.836,Z 792.613,A -85,B 0,C 180,E1 -21745.481,E2 -21745.481} C_VEL
LIN {X 0,Y 258.301,Z 779.528,A -85,B 0,C 180,E1 -21747.956,E2 -21747.956} C_VEL
LIN {X 0,Y 253.747,Z 769.908,A -85,B 0,C 180,E1 -21750.153,E2 -21750.153} C_VEL
LIN {X 0,Y 248.693,Z 760.026,A -85,B 0,C 180,E1 -21752.834,E2 -21752.834} C_VEL
LIN {X 0,Y 244.14,Z 753.181,A -85,B 0,C 180,E1 -21755.442,E2 -21755.442} C_VEL
LIN {X 0,Y 240.932,Z 748.601,A -85,B 0,C 180,E1 -21757.496,E2 -21757.496} C_VEL
LIN {X 0,Y 238.306,Z 744.992,A -85,B 0,C 180,E1 -21759.352,E2 -21759.352} C_VEL
LIN {X 0,Y 234.975,Z 740.519,A -85,B 0,C 180,E1 -21762.026,E2 -21762.026} C_VEL
LIN {X 0,Y 232.205,Z 736.889,A -85,B 0,C 180,E1 -21764.643,E2 -21764.643} C_VEL
LIN {X 0,Y 231.631,Z 735.881,A -85,B 0,C 180,E1 -21765.28,E2 -21765.28} C_VEL
LIN {X 0,Y 228.94,Z 732.999,A -85,B 0,C 180,E1 -21768.49,E2 -21768.49} C_VEL
LIN {X 0,Y 227.885,Z 730.704,A -85,B 0,C 180,E1 -21770.248,E2 -21770.248} C_VEL
LIN {X 0,Y 224.89,Z 727.161,A -85,B 0,C 180,E1 -21780,E2 -21780} C_VEL
LIN {X 0,Y 225.073,Z 728.238,A -85,B 0,C 180,E1 -21783.244,E2 -21783.244} C_VEL
LIN {X 0,Y 228.036,Z 731.003,A -85,B 0,C 180,E1 -21790.425,E2 -21790.425} C_VEL
LIN {X 0,Y 229.767,Z 734.173,A -85,B 0,C 180,E1 -21793.037,E2 -21793.037} C_VEL
LIN {X 0,Y 231.918,Z 736.236,A -85,B 0,C 180,E1 -21795.432,E2 -21795.432} C_VEL
LIN {X 0,Y 234.526,Z 740.074,A -85,B 0,C 180,E1 -21798,E2 -21798} C_VEL
LIN {X 0,Y 235.743,Z 741.471,A -85,B 0,C 180,E1 -21799.03,E2 -21799.03} C_VEL
LIN {X 0,Y 239.383,Z 746.411,A -85,B 0,C 180,E1 -21801.835,E2 -21801.835} C_VEL
LIN {X 0,Y 242.673,Z 751.117,A -85,B 0,C 180,E1 -21804.056,E2 -21804.056} C_VEL
LIN {X 0,Y 247.733,Z 758.382,A -85,B 0,C 180,E1 -21807.039,E2 -21807.039} C_VEL
LIN {X 0,Y 253.073,Z 766.875,A -85,B 0,C 180,E1 -21809.819,E2 -21809.819} C_VEL
LIN {X 0,Y 262.8,Z 781.018,A -85,B 0,C 180,E1 -21814.046,E2 -21814.046} C_VEL
LIN {X 0,Y 270.181,Z 789.531,A -85,B 0,C 180,E1 -21816.688,E2 -21816.688} C_VEL
LIN {X 0,Y 277.647,Z 796.953,A -85,B 0,C 180,E1 -21819.024,E2 -21819.024} C_VEL
LIN {X 0,Y 287.603,Z 805.412,A -85,B 0,C 180,E1 -21821.761,E2 -21821.761} C_VEL
LIN {X 0,Y 294.706,Z 811.394,A -85,B 0,C 180,E1 -21823.754,E2 -21823.754} C_VEL
LIN {X 0,Y 301.931,Z 817.496,A -85,B 0,C 180,E1 -21825.945,E2 -21825.945} C_VEL
LIN {X 0,Y 308.609,Z 823.293,A -85,B 0,C 180,E1 -21828.16,E2 -21828.16} C_VEL
LIN {X 0,Y 315.003,Z 828.807,A -85,B 0,C 180,E1 -21830.498,E2 -21830.498} C_VEL
LIN {X 0,Y 321.056,Z 833.867,A -85,B 0,C 180,E1 -21832.832,E2 -21832.832} C_VEL
LIN {X 0,Y 327.683,Z 839.609,A -85,B 0,C 180,E1 -21835.524,E2 -21835.524} C_VEL
LIN {X 0,Y 331.947,Z 843.195,A -85,B 0,C 180,E1 -21837.341,E2 -21837.341} C_VEL
LIN {X 0,Y 337.301,Z 847.705,A -85,B 0,C 180,E1 -21839.737,E2 -21839.737} C_VEL
LIN {X 0,Y 340.321,Z 850.023,A -85,B 0,C 180,E1 -21841.143,E2 -21841.143} C_VEL
LIN {X 0,Y 344.899,Z 854.008,A -85,B 0,C 180,E1 -21843.421,E2 -21843.421} C_VEL
LIN {X 0,Y 349.534,Z 857.173,A -85,B 0,C 180,E1 -21845.851,E2 -21845.851} C_VEL
LIN {X 0,Y 353.196,Z 860.487,A -85,B 0,C 180,E1 -21847.997,E2 -21847.997} C_VEL
LIN {X 0,Y 357.268,Z 863.553,A -85,B 0,C 180,E1 -21850.594,E2 -21850.594} C_VEL
LIN {X 0,Y 360.575,Z 865.617,A -85,B 0,C 180,E1 -21852.91,E2 -21852.91} C_VEL
LIN {X 0,Y 363.379,Z 868.362,A -85,B 0,C 180,E1 -21855.245,E2 -21855.245} C_VEL
LIN {X 0,Y 365.871,Z 870.268,A -85,B 0,C 180,E1 -21857.624,E2 -21857.624} C_VEL
LIN {X 0,Y 368.103,Z 871.631,A -85,B 0,C 180,E1 -21860.106,E2 -21860.106} C_VEL
LIN {X 0,Y 369.675,Z 872.346,A -85,B 0,C 180,E1 -21862.353,E2 -21862.353} C_VEL
LIN {X 0,Y 370.935,Z 872.93,A -85,B 0,C 180,E1 -21864.731,E2 -21864.731} C_VEL
LIN {X 0,Y 371.654,Z 873.296,A -85,B 0,C 180,E1 -21866.748,E2 -21866.748} C_VEL
LIN {X 0,Y 372.007,Z 873.444,A -85,B 0,C 180,E1 -21868.918,E2 -21868.918} C_VEL
LIN {X 0,Y 372.007,Z 873.444,A -85,B 0,C 180,E1 -21871.082,E2 -21871.082} C_VEL
LIN {X 0,Y 371.654,Z 873.298,A -85,B 0,C 180,E1 -21873.252,E2 -21873.252} C_VEL
LIN {X 0,Y 370.852,Z 872.873,A -85,B 0,C 180,E1 -21875.437,E2 -21875.437} C_VEL
LIN {X 0,Y 369.677,Z 872.334,A -85,B 0,C 180,E1 -21877.647,E2 -21877.647} C_VEL
LIN {X 0,Y 367.634,Z 871.37,A -85,B 0,C 180,E1 -21880.423,E2 -21880.423} C_VEL
LIN {X 0,Y 365.326,Z 869.894,A -85,B 0,C 180,E1 -21882.953,E2 -21882.953} C_VEL
LIN {X 0,Y 362.415,Z 867.505,A -85,B 0,C 180,E1 -21885.585,E2 -21885.585} C_VEL
LIN {X 0,Y 359.815,Z 864.956,A -85,B 0,C 180,E1 -21887.67,E2 -21887.67} C_VEL
LIN {X 0,Y 356.383,Z 862.924,A -85,B 0,C 180,E1 -21889.999,E2 -21889.999} C_VEL
LIN {X 0,Y 352.23,Z 859.67,A -85,B 0,C 180,E1 -21892.576,E2 -21892.576} C_VEL
LIN {X 0,Y 349.048,Z 856.832,A -85,B 0,C 180,E1 -21894.424,E2 -21894.424} C_VEL
LIN {X 0,Y 344.148,Z 853.43,A -85,B 0,C 180,E1 -21896.971,E2 -21896.971} C_VEL
LIN {X 0,Y 338.522,Z 848.55,A -85,B 0,C 180,E1 -21899.714,E2 -21899.714} C_VEL
LIN {X 0,Y 333.662,Z 844.726,A -85,B 0,C 180,E1 -21901.909,E2 -21901.909} C_VEL
LIN {X 0,Y 328.451,Z 840.227,A -85,B 0,C 180,E1 -21904.156,E2 -21904.156} C_VEL
LIN {X 0,Y 322.753,Z 835.327,A -85,B 0,C 180,E1 -21906.49,E2 -21906.49} C_VEL
LIN {X 0,Y 315.805,Z 829.53,A -85,B 0,C 180,E1 -21909.198,E2 -21909.198} C_VEL
LIN {X 0,Y 309.608,Z 824.131,A -85,B 0,C 180,E1 -21911.489,E2 -21911.489} C_VEL
LIN {X 0,Y 302.405,Z 817.898,A -85,B 0,C 180,E1 -21913.909,E2 -21913.909} C_VEL
LIN {X 0,Y 294.955,Z 811.581,A -85,B 0,C 180,E1 -21916.174,E2 -21916.174} C_VEL
LIN {X 0,Y 287.945,Z 805.703,A -85,B 0,C 180,E1 -21918.145,E2 -21918.145} C_VEL
LIN {X 0,Y 279.631,Z 798.685,A -85,B 0,C 180,E1 -21920.405,E2 -21920.405} C_VEL
LIN {X 0,Y 271.243,Z 790.685,A -85,B 0,C 180,E1 -21922.96,E2 -21922.96} C_VEL
LIN {X 0,Y 263.905,Z 782.337,A -85,B 0,C 180,E1 -21925.536,E2 -21925.536} C_VEL
LIN {X 0,Y 256.406,Z 772.138,A -85,B 0,C 180,E1 -21928.616,E2 -21928.616} C_VEL
LIN {X 0,Y 249.51,Z 761.141,A -85,B 0,C 180,E1 -21931.999,E2 -21931.999} C_VEL
LIN {X 0,Y 243.808,Z 752.723,A -85,B 0,C 180,E1 -21935.236,E2 -21935.236} C_VEL
LIN {X 0,Y 240.996,Z 748.719,A -85,B 0,C 180,E1 -21937.043,E2 -21937.043} C_VEL
LIN {X 0,Y 238.46,Z 745.138,A -85,B 0,C 180,E1 -21938.836,E2 -21938.836} C_VEL
LIN {X 0,Y 235.51,Z 741.055,A -85,B 0,C 180,E1 -21941.177,E2 -21941.177} C_VEL
LIN {X 0,Y 232.345,Z 737.09,A -85,B 0,C 180,E1 -21944.09,E2 -21944.09} C_VEL
LIN {X 0,Y 231.469,Z 735.709,A -85,B 0,C 180,E1 -21945.044,E2 -21945.044} C_VEL
LIN {X 0,Y 229.031,Z 733.115,A -85,B 0,C 180,E1 -21947.956,E2 -21947.956} C_VEL
LIN {X 0,Y 227.815,Z 730.663,A -85,B 0,C 180,E1 -21949.949,E2 -21949.949} C_VEL
LIN {X 0,Y 224.887,Z 727.308,A -85,B 0,C 180,E1 -21959.105,E2 -21959.105} C_VEL
LIN {X 0,Y 224.906,Z 727.354,A -85,B 0,C 180,E1 -21960.896,E2 -21960.896} C_VEL
LIN {X 0,Y 228.012,Z 730.918,A -85,B 0,C 180,E1 -21969.97,E2 -21969.97} C_VEL
LIN {X 0,Y 229.735,Z 734.14,A -85,B 0,C 180,E1 -21972.59,E2 -21972.59} C_VEL
LIN {X 0,Y 231.924,Z 736.307,A -85,B 0,C 180,E1 -21975.039,E2 -21975.039} C_VEL
LIN {X 0,Y 234.459,Z 740.029,A -85,B 0,C 180,E1 -21977.538,E2 -21977.538} C_VEL
LIN {X 0,Y 235.686,Z 741.437,A -85,B 0,C 180,E1 -21978.578,E2 -21978.578} C_VEL
LIN {X 0,Y 239.367,Z 746.42,A -85,B 0,C 180,E1 -21981.419,E2 -21981.419} C_VEL
LIN {X 0,Y 242.661,Z 751.058,A -85,B 0,C 180,E1 -21983.638,E2 -21983.638} C_VEL
LIN {X 0,Y 247.933,Z 758.727,A -85,B 0,C 180,E1 -21986.744,E2 -21986.744} C_VEL
LIN {X 0,Y 252.941,Z 768.247,A -85,B 0,C 180,E1 -21989.436,E2 -21989.436} C_VEL
LIN {X 0,Y 258.043,Z 778.915,A -85,B 0,C 180,E1 -21991.922,E2 -21991.922} C_VEL
LIN {X 0,Y 263.361,Z 791.453,A -85,B 0,C 180,E1 -21994.315,E2 -21994.315} C_VEL
LIN {X 0,Y 263.911,Z 792.79,A -85,B 0,C 180,E1 -21994.551,E2 -21994.551} C_VEL
LIN {X 0,Y 256.758,Z 889.086,A -85,B 0,C 180,E1 -21996.893,E2 -21996.893} C_VEL
LIN {X 0,Y 255.048,Z 902.613,A -85,B 0,C 180,E1 -21997.362,E2 -21997.362} C_VEL
LIN {X 0,Y 252.906,Z 914.738,A -85,B 0,C 180,E1 -21997.896,E2 -21997.896} C_VEL
LIN {X 0,Y 250.374,Z 926.16,A -85,B 0,C 180,E1 -21998.516,E2 -21998.516} C_VEL
LIN {X 0,Y 247.486,Z 937.541,A -85,B 0,C 180,E1 -21999.302,E2 -21999.302} C_VEL
LIN {X 0,Y 243.556,Z 950.771,A -85,B 0,C 180,E1 -22000.443,E2 -22000.443} C_VEL
LIN {X 0,Y 239.159,Z 963.501,A -85,B 0,C 180,E1 -22001.784,E2 -22001.784} C_VEL
LIN {X 0,Y 234.917,Z 974.49,A -85,B 0,C 180,E1 -22003.18,E2 -22003.18} C_VEL
LIN {X 0,Y 230.643,Z 984.781,A -85,B 0,C 180,E1 -22004.748,E2 -22004.748} C_VEL
LIN {X 0,Y 230.078,Z 986.07,A -85,B 0,C 180,E1 -22004.974,E2 -22004.974} C_VEL
LIN {X 0,Y 227.55,Z 990.76,A -85,B 0,C 180,E1 -22005.674,E2 -22005.674} C_VEL
LIN {X 0,Y 221.855,Z 997.991,A -85,B 0,C 180,E1 -22006.584,E2 -22006.584} C_VEL
LIN {X 0,Y 216.026,Z 1005.044,A -85,B 0,C 180,E1 -22007.599,E2 -22007.599} C_VEL
LIN {X 0,Y 213.299,Z 1009.008,A -85,B 0,C 180,E1 -22008.464,E2 -22008.464} C_VEL
LIN {X 0,Y 207.942,Z 1018.587,A -85,B 0,C 180,E1 -22011.144,E2 -22011.144} C_VEL
LIN {X 0,Y 202.34,Z 1028.201,A -85,B 0,C 180,E1 -22014.425,E2 -22014.425} C_VEL
LIN {X 0,Y 196.361,Z 1038.114,A -85,B 0,C 180,E1 -22018.738,E2 -22018.738} C_VEL
LIN {X 0,Y 191.994,Z 1045.38,A -85,B 0,C 180,E1 -22022.771,E2 -22022.771} C_VEL
LIN {X 0,Y 189.293,Z 1050.037,A -85,B 0,C 180,E1 -22025.896,E2 -22025.896} C_VEL
LIN {X 0,Y 186.499,Z 1055.145,A -85,B 0,C 180,E1 -22030.175,E2 -22030.175} C_VEL
LIN {X 0,Y 184.578,Z 1059.156,A -85,B 0,C 180,E1 -22034.542,E2 -22034.542} C_VEL
LIN {X 0,Y 183.435,Z 1062.127,A -85,B 0,C 180,E1 -22038.956,E2 -22038.956} C_VEL
LIN {X 0,Y 183.165,Z 1063.322,A -85,B 0,C 180,E1 -22041.172,E2 -22041.172} C_VEL
LIN {X 0,Y 182.977,Z 1064.806,A -85,B 0,C 180,E1 -22045.594,E2 -22045.594} C_VEL
LIN {X 0,Y 183.17,Z 1065.305,A -85,B 0,C 180,E1 -22050,E2 -22050} C_VEL
LIN {X 0,Y 182.977,Z 1064.806,A -85,B 0,C 180,E1 -22054.406,E2 -22054.406} C_VEL
LIN {X 0,Y 183.165,Z 1063.322,A -85,B 0,C 180,E1 -22058.828,E2 -22058.828} C_VEL
LIN {X 0,Y 183.862,Z 1060.836,A -85,B 0,C 180,E1 -22063.258,E2 -22063.258} C_VEL
LIN {X 0,Y 185.461,Z 1057.327,A -85,B 0,C 180,E1 -22067.647,E2 -22067.647} C_VEL
LIN {X 0,Y 187.777,Z 1052.738,A -85,B 0,C 180,E1 -22071.979,E2 -22071.979} C_VEL
LIN {X 0,Y 191.042,Z 1047.004,A -85,B 0,C 180,E1 -22076.196,E2 -22076.196} C_VEL
LIN {X 0,Y 193.975,Z 1042.085,A -85,B 0,C 180,E1 -22079.191,E2 -22079.191} C_VEL
LIN {X 0,Y 198.907,Z 1033.906,A -85,B 0,C 180,E1 -22083.206,E2 -22083.206} C_VEL
LIN {X 0,Y 203.131,Z 1026.923,A -85,B 0,C 180,E1 -22086.026,E2 -22086.026} C_VEL
LIN {X 0,Y 208.091,Z 1018.391,A -85,B 0,C 180,E1 -22088.907,E2 -22088.907} C_VEL
LIN {X 0,Y 212.868,Z 1009.848,A -85,B 0,C 180,E1 -22091.322,E2 -22091.322} C_VEL
LIN {X 0,Y 217.385,Z 1001.282,A -85,B 0,C 180,E1 -22093.392,E2 -22093.392} C_VEL
LIN {X 0,Y 223.325,Z 989.427,A -85,B 0,C 180,E1 -22095.719,E2 -22095.719} C_VEL
LIN {X 0,Y 227.784,Z 979.745,A -85,B 0,C 180,E1 -22097.319,E2 -22097.319} C_VEL
LIN {X 0,Y 232.8,Z 967.606,A -85,B 0,C 180,E1 -22098.999,E2 -22098.999} C_VEL
LIN {X 0,Y 237.29,Z 955.589,A -85,B 0,C 180,E1 -22100.358,E2 -22100.358} C_VEL
LIN {X 0,Y 241.285,Z 943.275,A -85,B 0,C 180,E1 -22101.515,E2 -22101.515} C_VEL
LIN {X 0,Y 244.785,Z 930.736,A -85,B 0,C 180,E1 -22102.478,E2 -22102.478} C_VEL
LIN {X 0,Y 247.94,Z 917.645,A -85,B 0,C 180,E1 -22103.248,E2 -22103.248} C_VEL
LIN {X 0,Y 250.53,Z 903.954,A -85,B 0,C 180,E1 -22103.879,E2 -22103.879} C_VEL
LIN {X 0,Y 252.292,Z 891.574,A -85,B 0,C 180,E1 -22104.309,E2 -22104.309} C_VEL
LIN {X 0,Y 254.442,Z 865.533,A -85,B 0,C 180,E1 -22104.997,E2 -22104.997} C_VEL
LIN {X 0,Y 259.684,Z 795.565,A -85,B 0,C 180,E1 -22106.68,E2 -22106.68} C_VEL
LIN {X 0,Y 254.246,Z 782.429,A -85,B 0,C 180,E1 -22109.279,E2 -22109.279} C_VEL
LIN {X 0,Y 248.58,Z 770.419,A -85,B 0,C 180,E1 -22112.25,E2 -22112.25} C_VEL
LIN {X 0,Y 245.191,Z 764.064,A -85,B 0,C 180,E1 -22114.194,E2 -22114.194} C_VEL
LIN {X 0,Y 239.778,Z 755.878,A -85,B 0,C 180,E1 -22117.602,E2 -22117.602} C_VEL
LIN {X 0,Y 236.319,Z 751.168,A -85,B 0,C 180,E1 -22120.114,E2 -22120.114} C_VEL
LIN {X 0,Y 233.389,Z 747.068,A -85,B 0,C 180,E1 -22122.587,E2 -22122.587} C_VEL
LIN {X 0,Y 230.759,Z 743.472,A -85,B 0,C 180,E1 -22125.194,E2 -22125.194} C_VEL
LIN {X 0,Y 230.169,Z 742.586,A -85,B 0,C 180,E1 -22125.861,E2 -22125.861} C_VEL
LIN {X 0,Y 227.636,Z 739.566,A -85,B 0,C 180,E1 -22129.087,E2 -22129.087} C_VEL
LIN {X 0,Y 226.758,Z 737.627,A -85,B 0,C 180,E1 -22130.635,E2 -22130.635} C_VEL
LIN {X 0,Y 224.023,Z 734.218,A -85,B 0,C 180,E1 -22140,E2 -22140} C_VEL
LIN {X 0,Y 226.87,Z 737.806,A -85,B 0,C 180,E1 -22149.971,E2 -22149.971} C_VEL
LIN {X 0,Y 228.732,Z 741.201,A -85,B 0,C 180,E1 -22152.871,E2 -22152.871} C_VEL
LIN {X 0,Y 230.594,Z 743.085,A -85,B 0,C 180,E1 -22155.014,E2 -22155.014} C_VEL
